(* PLC project BASIC, CODESYS CODESYS V3.5 SP16, author oscat *)
(* stored: creationDateTime 2020-05-24T16:39:18.0227817, version 3.31, modificationDateTime 2020-05-03T13:16:44.3823838, organization OSCAT *)
(* www.oscat.de *)

TYPE CALENDAR : STRUCT
  UTC : DT;  (* world time UTC *)
  YEAR : INT;  (* year of LDATE *)
  MONTH : INT;  (* month of LDATE *)
  DAY : INT;  (* day of LDATE *)
  WEEKDAY : INT;  (* weekday of LDATE *)
  OFFSET : INT;  (* Time Zone Offset for Local time in minutes *)
  DST_EN : BOOL;  (* daylight savings time enable *)
  DST_ON : BOOL;  (* true when daylight savings time os on *)
  NAME : STRING(5);  (* name of time zone *)
  LANGUAGE : INT;  (* location number pls see location setup *)
  LONGITUDE : REAL;  (* longitude of current location *)
  LATITUDE : REAL;  (* latitude of current location *)
  SUN_RISE : TOD;  (* sun_rise for current location *)
  SUN_SET : TOD;  (* sun_set for current location *)
  SUN_MIDDAY : TOD;  (* worldtime when sun stands at south position *)
  SUN_HEIGTH : REAL;  (* suns heigth at midday, south position *)
  SUN_HOR : REAL;  (* sun angle horizontal 0 = north in degrees *)
  SUN_VER : REAL;  (* sun angle vertical above horizon in degrees *)
  NIGHT : BOOL;  (* true between sun_set and sun_rise *)
  HOLIDAY : BOOL;  (* true when holiday *)
  HOLY_NAME : STRING(30);  (* name of holiday *)
  WORK_WEEK : INT;  (* current work week *)
END_STRUCT;
END_TYPE

TYPE COMPLEX : STRUCT
  re : REAL;
  im : REAL;
END_STRUCT;
END_TYPE

TYPE CONSTANTS_LANGUAGE : STRUCT
  DEFAULT : INT := 1;  (* 1=english, 2=german 3=french *)
  LMAX : INT := 3;
  WEEKDAYS : ARRAY[1..3, 1..7] OF STRING(10) := ['Monday', 'Tuesday', 'Wednesday', 'Thursday', 'Friday', 'Saturday', 'Sunday', 'Montag', 'Dienstag', 'Mittwoch', 'Donnerstag', 'Freitag', 'Samstag', 'Sonntag', 'Lundi', 'Mardi', 'Mercredi', 'Jeudi', 'Vendredi', 'Samedi', 'Dimanche'];
  WEEKDAYS2 : ARRAY[1..3, 1..7] OF STRING(2) := ['Mo', 'Tu', 'We', 'Th', 'Fr', 'Sa', 'Su', 'Mo', 'Di', 'Mi', 'Do', 'Fr', 'Sa', 'So', 'Lu', 'Ma', 'Me', 'Je', 'Ve', 'Sa', 'Di'];
  MONTHS : ARRAY[1..3, 1..12] OF STRING(10) := ['January', 'February', 'March', 'April', 'May', 'June', 'July', 'August', 'September', 'October', 'November', 'December', 'Januar', 'Februar', 'März', 'April', 'Mai', 'Juni', 'Juli', 'August', 'September', 'Oktober', 'November', 'Dezember', 'Janvier', 'Février', 'mars', 'Avril', 'Mai', 'Juin', 'Juillet', 'Août', 'Septembre', 'Octobre', 'Novembre', 'Decembre'];
  MONTHS3 : ARRAY[1..3, 1..12] OF STRING(3) := ['Jan', 'Feb', 'Mar', 'Apr', 'May', 'Jun', 'Jul', 'Aug', 'Sep', 'Oct', 'Nov', 'Dec', 'Jan', 'Feb', 'Mrz', 'Apr', 'Mai', 'Jun', 'Jul', 'Aug', 'Sep', 'Okt', 'Nov', 'Dez', 'Jan', 'Fev', 'Mar', 'Avr', 'Mai', 'Jun', 'Jul', 'Aou', 'Sep', 'Oct', 'Nov', 'Dec'];
  DIRS : ARRAY[1..3, 0..15] OF STRING(3) := ['N', 'NNE', 'NE', 'ENE', 'E', 'ESE', 'SE', 'SSE', 'S', 'SSW', 'SW', 'WSW', 'W', 'WNW', 'NW', 'NNW', 'N', 'NNO', 'NO', 'ONO', 'O', 'OSO', 'SO', 'SSO', 'S', 'SSW', 'SW', 'WSW', 'W', 'WNW', 'NW', 'NNW', 'N', 'NNO', 'NO', 'ONO', 'O', 'OSO', 'SO', 'SSO', 'S', 'SSW', 'SW', 'WSW', 'W', 'WNW', 'NW', 'NNW'];
END_STRUCT;
END_TYPE

TYPE CONSTANTS_LOCATION : STRUCT
  DEFAULT : INT := 1;  (* 1=germany, 2=austria 3=france 4=belgium-german 5= italien-Südtirol *)
  LMAX : INT := 5;
  LANGUAGE : ARRAY[1..5] OF INT := [2, 2, 3, 2, 2];  (* language spoken in the location *)
END_STRUCT;
END_TYPE

TYPE CONSTANTS_MATH : STRUCT
  PI : REAL := 3.1415926535897931;  (* Kreiszahl PI *)
  PI2 : REAL := 6.2831853071795862;  (* PI * 2 *)
  PI4 : REAL := 12.566370614359172;  (* PI * 4 *)
  PI05 : REAL := 1.5707963267949;  (* PI / 2 *)
  PI025 : REAL := 0.785398163397448;  (* PI / 4 *)
  PI_INV : REAL := 0.318309886183791;  (* 1 / PI *)
  E : REAL := 2.7182818284590451;  (* Eulersche Konstante e *)
  E_INV : REAL := 0.367879441171442;  (* 1 / e *)
  SQ2 : REAL := 1.4142135623731;  (* Wurzel von 2 *)
END_STRUCT;
END_TYPE

TYPE CONSTANTS_PHYS : STRUCT
  C : REAL := 299792458;  (* Lichtgeschwindigkeit in m/s *)
  E : REAL := 1.60217653E-19;  (* elementarladung in Colomb = A * s *)
  G : REAL := 9.80665;  (* Erdbeschleunigung in m / s² *)
  T0 : REAL := -273.15;  (* absoluter Nullpunkt in °C *)
  RU : REAL := 8.314472;  (* Universelle Gaskonstante in J / (mol · K) *)
  PN : REAL := 101325;  (* NormalDruck in Pa *)
END_STRUCT;
END_TYPE

TYPE CONSTANTS_SETUP : STRUCT
  EXTENDED_ASCII : BOOL := TRUE;  (* setup Parameters *)
  CHARNAMES : ARRAY[1..4] OF STRING(253) := [';"&quot;&&amp;<&lt;>&gt;&euro; &nbsp;¡&iexcl;¢&cent;£&pound;¤&curren;¥&yen;¦&brvbar;§&sect;¨&uml;©&copy;ª&ordf;«&laquo;¬&not;­&shy;®&reg;¯&macr;°&deg;±&plusmn;²&sup2;³&sup3;´&acute;µ&micro;¶&para;·&middot;¸&cedil;¹&sup1;º&ordm;»&raquo;¼&frac14;Û&Ucirc;', ';¾&frac34;¿&iquest;À&Agrave;Á&Aacute;Â&Acirc;Ã&Atilde;Ä&Auml;Å&Aring;Æ&AElig;Ç&Ccedil;È&Egrave;É&Eacute;Ê&Ecirc;Ë&Euml;Ì&Igrave;Í&Iacute;Î&Icirc;Ï&Iuml;Ð&ETH;Ñ&Ntilde;Ò&Ograve;Ó&Oacute;Ô&Ocirc;Õ&Otilde;Ö&Ouml;×&times;Ø&Oslash;Ù&Ugrave;Ú&Uacute;½&frac12;', ';Ü&Uuml;Ý&Yacute;Þ&THORN;ß&szlig;à&agrave;á&aacute;â&acirc;ã&atilde;ä&auml;å&aring;æ&aelig;ç&ccedil;è&egrave;é&eacute;ê&ecirc;ë&euml;ì&igrave;í&iacute;î&icirc;ï&iuml;ð&eth;ñ&ntilde;ò&ograve;ó&oacute;ô&ocirc;õ&otilde;ö&ouml;÷&divide;ø&oslash;ù&ugrave;', ';ú&uacute;û&ucirc;ü&uuml;ý&yacute;þ&thorn;ÿ&yuml;'];
  MTH_OFS : ARRAY[1..12] OF INT := [0, 31, 59, 90, 120, 151, 181, 212, 243, 273, 304, 334];
  DECADES : ARRAY[0..8] OF REAL := [1, 10, 100, 1000, 10000, 10000, 100000, 1000000, 10000000];
END_STRUCT;
END_TYPE

TYPE ESR_DATA : STRUCT
  TYP : BYTE;
  ADRESS : STRING(10);
  DS : DT;
  TS : TIME;
  DATA : ARRAY[0..7] OF BYTE;
END_STRUCT;
END_TYPE

TYPE FRACTION : STRUCT
  NUMERATOR : INT;
  DENOMINATOR : INT;
END_STRUCT;
END_TYPE

TYPE HOLIDAY_DATA : STRUCT
  NAME : STRING(30);
  DAY : SINT;
  MONTH : SINT;
  USE : SINT;
END_STRUCT;
END_TYPE

TYPE REAL2 : STRUCT
  R1 : REAL;  (* small value *)
  RX : REAL;  (* big value *)
END_STRUCT;
END_TYPE

TYPE SDT : STRUCT
  YEAR : INT;
  MONTH : INT;
  DAY : INT;
  WEEKDAY : INT;
  HOUR : INT;
  MINUTE : INT;
  SECOND : INT;
  MS : INT;
END_STRUCT;
END_TYPE

TYPE TIMER_EVENT : STRUCT
  TYP : BYTE;
  CHANNEL : BYTE;
  DAY : BYTE;
  START : TOD;
  DURATION : TIME;
  LAND : BYTE;
  LOR : BYTE;
  LAST : DT;
END_STRUCT;
END_TYPE

TYPE VECTOR_3 : STRUCT
  X : REAL;
  Y : REAL;
  Z : REAL;
END_STRUCT;
END_TYPE

VAR_GLOBAL CONSTANT  (* Constants *)
  STRING_LENGTH : INT := 250;
  LIST_LENGTH : INT := 250;
END_VAR

VAR_GLOBAL  (* Globale_Variablen *)
  MATH : CONSTANTS_MATH;
  PHYS : CONSTANTS_PHYS;
  LANGUAGE : CONSTANTS_LANGUAGE;
  SETUP : CONSTANTS_SETUP;
  LOCATION : CONSTANTS_LOCATION;
END_VAR


FUNCTION _BUFFER_CLEAR : BOOL
  VAR_INPUT
    PT : POINTER TO BYTE;
    SIZE : UINT;
  END_VAR
  VAR
    ptw : POINTER TO DWORD;
    temp : DWORD;
    end : DWORD;
    end32 : DWORD;
  END_VAR

            (* this routine uses 32 bit access to gain speed *)
(* first access bytes till pointer is aligned for 32 bit access *)
temp := pt;
end := temp + UINT_TO_DWORD(size);
end32 := end - 3;
WHILE (pt < end) AND ((temp AND 16#00000003) > 0) DO
	pt^ := 0;
	pt := pt + 1;
	temp := temp + 1;
END_WHILE;
(* pointer is aligned, now copy 32 bits at a time *)
ptw := pt;
WHILE ptw < end32 DO (* *)
	ptw^ := 0;
	ptw := ptw + 4;
END_WHILE;
(* copy the remaining bytes in byte mode *)
pt := ptw;
WHILE pt < end DO
	pt^ := 0;
	pt := pt + 1;
END_WHILE;

_BUFFER_CLEAR := TRUE;

(* revision History
hm 	5. mar. 2008	rev 1.0
	original version

hm	16. mar. 2008	rev 1.1
	added type conversion to avoid warnings under codesys 30
	chaged type of input size to uint
	deleted unused variable i

hm	31. oct. 2008	rev 1.2
	corrected an error while routine would write outside of arrays

*)
          
END_FUNCTION

FUNCTION _BUFFER_INIT : BOOL
  VAR_INPUT
    PT : POINTER TO BYTE;
    SIZE : UINT;
    INIT : BYTE;
  END_VAR
  VAR
    ptw : POINTER TO DWORD;
    temp : DWORD;
    end : DWORD;
    end32 : DWORD;
  END_VAR

            (* this routine uses 32 bit access to gain speed *)
(* first access bytes till pointer is aligned for 32 bit access *)
temp := pt;
end := temp + UINT_TO_DWORD(size);
end32 := end - 3;
WHILE (pt < end) AND ((temp AND 16#00000003) > 0) DO
	pt^ := init;
	pt := pt + 1;
	temp := temp + 1;
END_WHILE;
(* pointer is aligned, now copy 32 bits at a time *)
ptw := pt;
temp := SHL(BYTE_TO_DWORD(init),24) OR SHL(BYTE_TO_DWORD(init),16) OR SHL(BYTE_TO_DWORD(init),8) OR BYTE_TO_DWORD(init);
WHILE ptw < end32 DO
	ptw^ := temp;
	ptw := ptw + 4;
END_WHILE;
(* copy the remaining bytes in byte mode *)
pt := ptw;
WHILE pt < end DO
	pt^ := init;
	pt := pt + 1;
END_WHILE;

_BUFFER_INIT := TRUE;

(* revision History
hm 	5. mar. 2008	rev 1.0
	original version

hm	16. mar. 2008	rev 1.1
	added type conversion to avoid warnings under codesys 3.0
	chaged type of input size to uint.

hm	31. oct. 2008	rev 1.2
	corrected an error while routine would write outside of arrays

*)
          
END_FUNCTION

FUNCTION _BUFFER_INSERT : BOOL
  VAR_INPUT
    STR : STRING(STRING_LENGTH);
    POS : INT;
    PT : POINTER TO ARRAY[0..32767] OF BYTE;
    SIZE : UINT;
  END_VAR
  VAR
    end : INT;
    lx : INT;
    i : INT;
  END_VAR

            lx := LEN(str);
end := pos + lx;
(* first move the upper part of the buffer to make space for the string *)
FOR i := UINT_TO_INT(size) - 1 TO end BY -1 DO
	pt^[i] := pt^[i-lx];
END_FOR;
(* copy the string *)
_BUFFER_INSERT := _STRING_TO_BUFFER(str, pos, PT, size);


(* revision History
hm 	9. mar. 2008	rev 1.0
	original version

hm	16. mar. 2008	rev 1.1
	changed type of input size to uint

hm	13. may. 2008	rev 1.2
	changed type of pointer to array[1..32767]
	changed size of string to STRING_LENGTH

hm	23. mar. 2009	rev 1.3
	avoid writing to input pos

hm	12. nov. 2009	rev 1.4
	code optimized

*)
          
END_FUNCTION

FUNCTION _BUFFER_UPPERCASE : BOOL
  VAR_INPUT
    PT : POINTER TO ARRAY[0..32000] OF BYTE;
    SIZE : INT;
  END_VAR
  VAR
    pos : INT;
  END_VAR

            pos := 0;
WHILE pos < size DO
	PT^[pos] := TO_UPPER(pt^[pos]);
	pos := pos + 1;
END_WHILE;

_BUFFER_UPPERCASE := TRUE;

(* revision History
hm 	20. jan. 2011	rev 1.0
	original version

*)
          
END_FUNCTION

FUNCTION _STRING_TO_BUFFER : BOOL
  VAR_INPUT
    STR : STRING(STRING_LENGTH);
    POS : INT;
    PT : POINTER TO ARRAY[0..32767] OF BYTE;
    SIZE : UINT;
  END_VAR
  VAR
    ps : POINTER TO BYTE;
    i : INT;
    end : INT;
  END_VAR

            ps := ADR(str);
end := MIN(pos + LEN(str), UINT_TO_INT(size));
IF end > 0 THEN end := end -1; END_IF;
FOR i := pos TO end DO
	pt^[i] := ps^;
	ps := ps + 1;
END_FOR;

_STRING_TO_BUFFER := TRUE;

(* revision History

hm 	5. mar. 2008	rev 1.0
	original version

hm	16. mar. 2008	rev 1.1
	changed type of input size to uint

hm	13. may. 2008	rev 1.2
	changed type of pointer to array[1..32767]
	changed size of string to STRING_LENGTH

hm	12. nov. 2009	rev 1.3
	limit end to size - 1

*)
          
END_FUNCTION

FUNCTION BUFFER_COMP : INT
  VAR_INPUT
    PT1 : POINTER TO ARRAY[0..32767] OF BYTE;
    SIZE1 : INT;
    PT2 : POINTER TO ARRAY[0..32767] OF BYTE;
    SIZE2 : INT;
    START : INT;
  END_VAR
  VAR
    i : INT;
    j : INT;
    end : INT;
    firstbyte : BYTE;
  END_VAR

            (* search for first character match *)
IF size2 <= size1 THEN
	end := size1 - size2;
	firstbyte := PT2^[0];
	FOR i := START TO end DO
		IF PT1^[i] = firstbyte THEN
			(* first character matches, now compare rest of array *)
			j := 1;
			WHILE j < size2 DO
				IF pt2^[j] <> pt1^[j+i] THEN EXIT; END_IF;
				j := j + 1;
			END_WHILE;
			(* when J > size2 a match was found return the position i in buffer1 *)
			IF j = size2 THEN
				BUFFER_COMP := i;
				RETURN;
			END_IF;
		END_IF;
	END_FOR;
END_IF;
BUFFER_COMP := -1;


(*
hm 14. nov. 2008	rev 1.0
	original version

hm	12. nov. 2009	rev 1.1
	performance increase

*)
          
END_FUNCTION

FUNCTION BUFFER_SEARCH : INT
  VAR_INPUT
    PT : POINTER TO ARRAY[0..32767] OF BYTE;
    SIZE : INT;
    STR : STRING(STRING_LENGTH);
    POS : INT;
    IGN : BOOL;
  END_VAR
  VAR
    ps : POINTER TO ARRAY[0..STRING_LENGTH] OF BYTE;
    chx : BYTE;
    i : INT;
    end : INT;
    k : INT;
    lx : INT;
  END_VAR

            ps := ADR(STR);
lx := LEN(STR);
end := MIN(SIZE - lx, SIZE - 1);
lx := lx - 1;
FOR i := pos TO end DO
	FOR k := 0 TO lx DO
		IF IGN THEN chx := TO_UPPER(pt^[i+k]); ELSE chx := pt^[i+k]; END_IF;
		IF ps^[k] <> chx THEN EXIT; END_IF;
	END_FOR;
	IF k > lx THEN
		BUFFER_SEARCH := i;
		RETURN;
	END_IF;
END_FOR;
BUFFER_SEARCH := -1;


(* revision History

hm 5. mar. 2008	rev 1.0
	original version

hm	16. mar. 2008	rev 1.1
	chaged type of input size to uint

hm	13. may. 2008	rev 1.2
	changed type of pointer to array[1..32767]
	changed size of string to STRING_LENGTH

hm	12. nov. 2009	rev 1.3
	limit end to array size

hm	25. jan. 2011	rev 1.4
	ign = True will now ignore case
	return -1 if nothing found
*)
          
END_FUNCTION

FUNCTION BUFFER_TO_STRING : STRING(STRING_LENGTH)
  VAR_INPUT
    PT : POINTER TO ARRAY[0..32767] OF BYTE;
    SIZE : UINT;
    START : UINT;
    STOP : UINT;
  END_VAR
  VAR
    ps : POINTER TO BYTE;
    i : UINT;
    stp : UINT;
    sta : UINT;
  END_VAR

            ps := ADR(BUFFER_TO_STRING);
IF size = 0 THEN RETURN; END_IF;
sta := MIN(start, size -1);
stp := MIN(stop, size -1);

(* check for maximum string_length *)
IF UINT_TO_INT(stp - sta + 1) >= STRING_LENGTH THEN
	stp := sta + INT_TO_UINT(STRING_LENGTH) - 1;
END_IF;

FOR i := sta TO stp DO
	ps^ := pt^[i];
	ps := ps + 1;
END_FOR;

(* terminate the string *)

ps^ := 0;



(* revision History
hm 	5. mar. 2008	rev 1.0
	original version

hm	16. mar. 2008	rev 1.1
	changed type of input size to uint

hm	13. may. 2008	rev 1.2
	changed type of pointer to array[0..32767]
	changed size of string to STRING_LENGTH

hm	12. jun. 2008	rev 1.3
	check for pointer overrun
	change input start and stop to uint
	added type conversions to avoid warnings under codesys 3.0

hm	23. mar. 2009	rev 1.4
	avoid writing to input stop

hm	12. nov. 2009 rev 1.5
	limit start and stop to size -1

*)
          
END_FUNCTION

FUNCTION_BLOCK DRIVER_1
  VAR_INPUT
    {attribute 'input_constant'}
    Toggle_Mode : BOOL;
    {attribute 'input_constant'}
    Timeout : TIME;
    SET : BOOL;
    IN : BOOL;
    RST : BOOL;
  END_VAR
  VAR_OUTPUT
    Q : BOOL;
  END_VAR
  VAR
    off : TON;
    edge : BOOL;
  END_VAR

            IF off.Q THEN Q := FALSE; END_IF;
IF rst THEN
	Q := FALSE;
ELSIF set THEN
	Q := TRUE;
ELSIF IN AND NOT edge THEN
	IF toggle_mode THEN q := NOT Q; ELSE q := TRUE; END_IF;
END_IF;
edge := in;
IF timeout > t#0s THEN off(in := Q, PT := Timeout); END_IF;


(* revision history
hm	2. jan 2008		rev 1.0
	original version

*)
          
END_FUNCTION_BLOCK

FUNCTION_BLOCK DRIVER_4
  VAR_INPUT
    {attribute 'input_constant'}
    Toggle_Mode : BOOL;
    {attribute 'input_constant'}
    Timeout : TIME;
    SET : BOOL;
    IN0 : BOOL;
    IN1 : BOOL;
    IN2 : BOOL;
    IN3 : BOOL;
    RST : BOOL;
  END_VAR
  VAR_OUTPUT
    Q0 : BOOL;
    Q1 : BOOL;
    Q2 : BOOL;
    Q3 : BOOL;
  END_VAR
  VAR
    d0 : DRIVER_1;
    d1 : DRIVER_1;
    d2 : DRIVER_1;
    d3 : DRIVER_1;
  END_VAR

            D0(Set:=set, in:=in0, rst:=rst, toggle_mode:=toggle_mode, timeout:=timeout);
D1(Set:=set, in:=in1, rst:=rst, toggle_mode:=toggle_mode, timeout:=timeout);
D2(Set:=set, in:=in2, rst:=rst, toggle_mode:=toggle_mode, timeout:=timeout);
D3(Set:=set, in:=in3, rst:=rst, toggle_mode:=toggle_mode, timeout:=timeout);
Q0 := D0.Q;
Q1 := D1.Q;
Q2 := D2.Q;
Q3 := D3.Q;


(* revision history
hm	2. jan 2008		rev 1.0
	original version

*)
          
END_FUNCTION_BLOCK

FUNCTION_BLOCK DRIVER_4C
  VAR_INPUT
    IN : BOOL;
    RST : BOOL;
    {attribute 'input_constant'}
    Timeout : TIME;
    {attribute 'input_constant'}
    SX : ARRAY[1..7] OF BYTE := [1, 3, 7, 15];
  END_VAR
  VAR_OUTPUT
    SN : INT;
    Q0 : BOOL;
    Q1 : BOOL;
    Q2 : BOOL;
    Q3 : BOOL;
  END_VAR
  VAR
    off : TON;
    edge : BOOL;
  END_VAR

            IF RST OR off.Q THEN
	SN := 0;
ELSIF IN AND NOT edge THEN
	SN := SN + 1;
	IF SN > 7 OR SX[SN] = 0 THEN SN := 0; END_IF;
END_IF;
edge := in;
IF SN > 0 THEN
	Q0 := SX[SN].0;
	Q1 := SX[SN].1;
	Q2 := SX[SN].2;
	Q3 := SX[SN].3;
ELSE
	Q0 := FALSE;
	Q1 := FALSE;
	Q2 := FALSE;
	Q3 := FALSE;
END_IF;

(* maximaum timeout *)
IF timeout > t#0s THEN off(in := SN > 0, PT := Timeout); END_IF;


(* revision history
hm	23. mar. 2009	rev 1.0
	original version

*)
          
END_FUNCTION_BLOCK

FUNCTION_BLOCK FLOW_CONTROL
  VAR_INPUT
    IN : BOOL;
    REQ : BOOL;
    ENQ : BOOL;
    RST : BOOL;
    {attribute 'input_constant'}
    T_AUTO : TIME := TIME#60m0s0ms;
    {attribute 'input_constant'}
    T_DELAY : TIME := TIME#1380m0s0ms;
  END_VAR
  VAR_OUTPUT
    Q : BOOL;
    STATUS : BYTE;
  END_VAR
  VAR
    timer : TP_1D;
  END_VAR

            STATUS := 100;
IF RST THEN
	Q := FALSE;
	timer(rst := TRUE);
	timer.RST := FALSE;
	STATUS := 103;
ELSIF ENQ THEN
	IF IN THEN
		status := 101;
	END_IF;
	IF REQ THEN
		(* timer will generate a timed pulse after TP goes high *)
		timer.PT1 := T_AUTO;
		timer.PTD := T_DELAY;
		timer.IN := TRUE;
		STATUS := 102;
	END_IF;
END_IF;


(* set output and run timer *)
timer();
timer.IN := FALSE;
Q := (IN AND ENQ) OR timer.Q;



(* revision history
hm 	28. jun. 2008 	rev 1.0
	original version

*)
          
END_FUNCTION_BLOCK

FUNCTION_BLOCK FT_Profile
  VAR_INPUT
    K : REAL := 1;
    O : REAL;
    M : REAL := 1;
    E : BOOL;
    {attribute 'input_constant'}
    value_0 : REAL;
    {attribute 'input_constant'}
    time_1 : TIME;
    {attribute 'input_constant'}
    value_1 : REAL;
    {attribute 'input_constant'}
    time_2 : TIME;
    {attribute 'input_constant'}
    value_2 : REAL;
    {attribute 'input_constant'}
    time_3 : TIME;
    {attribute 'input_constant'}
    value_3 : REAL;
    {attribute 'input_constant'}
    time_10 : TIME;
    {attribute 'input_constant'}
    value_10 : REAL;
    {attribute 'input_constant'}
    time_11 : TIME;
    {attribute 'input_constant'}
    value_11 : REAL;
    {attribute 'input_constant'}
    time_12 : TIME;
    {attribute 'input_constant'}
    value_12 : REAL;
    {attribute 'input_constant'}
    time_13 : TIME;
    {attribute 'input_constant'}
    value_13 : REAL;
  END_VAR
  VAR_OUTPUT
    Y : REAL;
    RUN : BOOL;
    ET : TIME;
  END_VAR
  VAR
    tx : TIME;
    edge : BOOL;
    state : BYTE;
    ta : TIME;
    tb : TIME;
    t0 : TIME;
    temp : REAL;
    va : REAL;
    vb : REAL;
  END_VAR

            (* read system time *)
tx := DWORD_TO_TIME(T_PLC_MS());

(* determine start condition *)
IF E AND NOT edge THEN
	RUN := TRUE;
	ET := t#0s;
	t0 := tx;
	ta := tx;
	tb := multime(time_1, M);
	va := value_0;
	vb := value_1;
	temp := value_0;
	state := 1;
END_IF;
edge := E;

(* generate startup profile *)
IF run THEN
	CASE state OF
		1:	IF tx - ta >= tb THEN
				ta := ta + tb;
				tb := multime(time_2 - time_1, M);
				va := value_1;
				vb := value_2;
				temp := value_1;
				state := 2;
			ELSE
				temp := ((vb - va) * TIME_TO_REAL(tx - ta) / TIME_TO_REAL(tb) + va);
			END_IF;
		2:	IF tx - ta >= tb THEN
				ta := ta + tb;
				tb := multime(time_3 - time_2, M);
				va := value_2;
				vb := value_3;
				temp := value_2;
				state := 3;
			ELSE
				temp := ((vb - va) * TIME_TO_REAL(tx - ta) / TIME_TO_REAL(tb) + va);
			END_IF;
		3:	IF tx - ta >= tb THEN
				ta := ta + tb;
				tb := multime(time_10 - time_3, M);
				va := value_3;
				vb := value_10;
				temp := value_3;
				state := 4;
			ELSE
				temp := ((vb - va) * TIME_TO_REAL(tx - ta) / TIME_TO_REAL(tb) + va);
			END_IF;
		4 :	IF tx - ta >= tb THEN
				ta := ta + tb;
				tb := multime(time_11 - time_10, M);
				va := value_10;
				vb := value_11;
				temp := value_10;
				IF E THEN state := 5; ELSE state := 6; END_IF;
			ELSE
				temp := ((vb - va) * TIME_TO_REAL(tx - ta) / TIME_TO_REAL(tb) + va);
			END_IF;
		5:	(* extend the signal while E is true *)
			IF E THEN
				ta := tx;
			ELSE
				state := 6;
			END_IF;
		6:	IF tx - ta >= tb THEN
				ta := ta + tb;
				tb := multime(time_12 - time_11, M);
				va := value_11;
				vb := value_12;
				temp := value_11;
				state := 7;
			ELSE
				temp := ((vb - va) * TIME_TO_REAL(tx - ta) / TIME_TO_REAL(tb) + va);
			END_IF;
		7:	IF tx - ta >= tb THEN
				ta := ta + tb;
				tb := multime(time_13 - time_12, M);
				va := value_12;
				vb := value_13;
				temp := value_12;
				state := 8;
			ELSE
				temp := ((vb - va) * TIME_TO_REAL(tx - ta) / TIME_TO_REAL(tb) + va);
			END_IF;
		8:	IF tx - ta >= tb THEN
				temp := value_13;
				run := FALSE;
			ELSE
				temp := ((vb - va) * TIME_TO_REAL(tx - ta) / TIME_TO_REAL(tb) + va);
			END_IF;
	END_CASE;
	Y := temp * K + O;
	ET := tx - t0;
END_IF;

(* revision history
hm	27 feb 2007		rev 1.0
	original version

hm	15. sep2007		rev 1.1
	replaced Time() with T_PLC_MS for compatibility and performance reasons

*)
          
END_FUNCTION_BLOCK

FUNCTION_BLOCK INC_DEC
  VAR_INPUT
    CHa : BOOL;
    CHb : BOOL;
    RST : BOOL;
  END_VAR
  VAR_OUTPUT
    dir : BOOL;
    cnt : INT;
  END_VAR
  VAR
    edgea : BOOL;
    clk : BOOL;
    clka : BOOL;
    clkb : BOOL;
    edgeb : BOOL;
    axb : BOOL;
  END_VAR

            axb := cha XOR chb;

(* create pulses for channel a *)
clka := cha XOR edgea;
edgea := cha;

clkb := chb XOR edgeb;
edgeb := chb;

(* create pulses for both channels *)
clk := clka OR clkb;

(* set the direction output *)
IF axb AND clka THEN dir := TRUE; END_IF;
IF axb AND clkb THEN dir := FALSE; END_IF;

(* increment or decrement the counter *)
IF clk AND dir THEN cnt := cnt + 1; END_IF;
IF clk AND NOT dir THEN cnt := cnt -1; END_IF;

(* reset the counter if rst active *)
IF rst THEN cnt := 0; END_IF;

          
END_FUNCTION_BLOCK

FUNCTION_BLOCK INTERLOCK
  VAR_INPUT
    I1 : BOOL;
    I2 : BOOL;
    TL : TIME;
  END_VAR
  VAR_OUTPUT
    Q1 : BOOL;
    Q2 : BOOL;
  END_VAR
  VAR
    T1 : TOF;
    T2 : TOF;
  END_VAR

            (* the input signal have a run delay to lockout the other input *)
T1(IN := I1, PT := TL);
T2(IN := I2, PT := TL);

Q1 := I1 AND NOT t2.Q;
Q2 := I2 AND NOT t1.Q;


(* revision history

hm	28 sep 2007		rev 1.0
	original version

*)
          
END_FUNCTION_BLOCK

FUNCTION_BLOCK INTERLOCK_4
  VAR_INPUT
    I0 : BOOL;
    I1 : BOOL;
    I2 : BOOL;
    I3 : BOOL;
    E : BOOL;
    MODE : INT;
  END_VAR
  VAR_OUTPUT
    OUT : BYTE;
    TP : BOOL;
  END_VAR
  VAR
    in : BYTE;
    last : BYTE;
    old : BYTE;
    lmode : INT;
  END_VAR

            (* check if enable is active *)
IF E THEN
(* reset all vars when there is a mode change on thy fly *)
	IF mode <> lmode THEN
		out := 0;
		last := 0;
		old := 0;
		lmode := mode;
	END_IF;
	(* load inputs into in *)
	in.0 := I0;
	in.1 := I1;
	in.2 := I2;
	in.3 := I3;
	(* only execute when there is any change *)
	IF in <> last THEN
		(* only execute when inputs have chages state *)
		CASE mode OF
			0:	(* output directly display inputs as bits in byte out *)
				out := in;

			1:	(* the input with the highest number will be acepted *)
				IF in.3 THEN out := 8;
				ELSIF in.2 THEN out := 4;
				ELSIF in.1 THEN out := 2;
				ELSE out := in;
				END_IF;

			2:	(* input last pressed will be displayed only *)
				last := ((in XOR last) AND in);
				IF last.3 THEN out := 8;
				ELSIF last.2 THEN out := 4;
				ELSIF last.1 THEN out := 2;
				ELSE out := last;
				END_IF;

			3:	(* any input active will disable all other inputs *)
				IF (out AND in) = 0 THEN
					IF in.3 THEN out := 8;
					ELSIF in.2 THEN out := 4;
					ELSIF in.1 THEN out := 2;
					ELSE out := in;
					END_IF;
				END_IF;

		END_CASE;
		last := in;
	END_IF;
	tp := out <> old;
	old := out;
ELSE
	out := 0;
	last := 0;
	old := 0;
	lmode := 0;
	tp := FALSE;
END_IF;


(* revision history
hm	24. oct 2008	rev 1.0
	original version

hm	14. mar. 2009	rev 1.1
	replaced double assignments

*)
          
END_FUNCTION_BLOCK

FUNCTION MANUAL : BOOL
  VAR_INPUT
    IN : BOOL;
    ON : BOOL;
    OFF : BOOL;
  END_VAR

            MANUAL := NOT OFF AND (IN OR ON);



(* revision history
hm	21. nov 2008	rev 1.0
	original version


*)
          
END_FUNCTION

FUNCTION_BLOCK MANUAL_1
  VAR_INPUT
    IN : BOOL;
    MAN : BOOL;
    M_I : BOOL;
    SET : BOOL;
    RST : BOOL;
  END_VAR
  VAR_OUTPUT
    Q : BOOL;
    STATUS : BYTE;
  END_VAR
  VAR
    S_edge : BOOL;
    r_edge : BOOL;
    edge : BOOL;
  END_VAR

            IF NOT man THEN
	Q := IN;
	STATUS := 100;
	edge := FALSE;
ELSIF NOT s_edge AND set THEN
	Q := TRUE;
	edge := TRUE;
	status := 101;
ELSIF NOT r_edge AND rst THEN
	Q := FALSE;
	edge := TRUE;
	status := 102;
ELSIF NOT edge THEN
	Q := M_I;
	status := 103;
END_IF;

(* remember levels of manual signals *)
s_edge := SET;
r_edge := RST;



(* revision history
hm	17. jun 2008	rev 1.0
	original version

hm	17. oct 2008	rev 1.1
	deleted unnecessary variable m_edge

hm	14. mar. 2009	rev 1.2
	replaced double assignments

*)
          
END_FUNCTION_BLOCK

FUNCTION_BLOCK MANUAL_2
  VAR_INPUT
    IN : BOOL;
    ENA : BOOL;
    ON : BOOL;
    OFF : BOOL;
    MAN : BOOL;
  END_VAR
  VAR_OUTPUT
    Q : BOOL;
    STATUS : BYTE;
  END_VAR

            IF ena THEN
	IF NOT ON AND NOT OFF THEN
		Q := IN;
		STATUS := 100;
	ELSIF on AND NOT off THEN
		Q := TRUE;
		STATUS := 101;
	ELSIF NOT on AND off THEN
		q := FALSE;
		STATUS := 102;
	ELSE
		Q := MAN;
		STATUS := 103;
	END_IF;
ELSE
	Q := FALSE;
	STATUS := 104;
END_IF;



(* revision history
hm	22. sep. 2008		rev 1.0
	original version

*)
          
END_FUNCTION_BLOCK

FUNCTION_BLOCK MANUAL_4
  VAR_INPUT
    I0 : BOOL;
    I1 : BOOL;
    I2 : BOOL;
    I3 : BOOL;
    MAN : BOOL;
    STP : BOOL;
    M0 : BOOL;
    M1 : BOOL;
    M2 : BOOL;
    M3 : BOOL;
  END_VAR
  VAR_OUTPUT
    Q0 : BOOL;
    Q1 : BOOL;
    Q2 : BOOL;
    Q3 : BOOL;
    STATUS : BYTE;
  END_VAR
  VAR
    edge : BOOL;
    pos : INT;
    tog : BOOL;
  END_VAR

            IF man THEN
	IF NOT TOG THEN
		Q0 := M0;
		Q1 := M1;
		Q2 := M2;
		Q3 := M3;
		STATUS := 101;
	END_IF;
	IF STP AND NOT edge THEN
		tog := TRUE;
		CASE pos OF
			0:	Q0 := TRUE;
				Q1 := FALSE;
				Q2 := FALSE;
				Q3 := FALSE;
				STATUS := 110;
			1:	Q0 := FALSE;
				Q1 := TRUE;
				Q2 := FALSE;
				Q3 := FALSE;
				STATUS := 111;
			2:	Q0 := FALSE;
				Q1 := FALSE;
				Q2 := TRUE;
				Q3 := FALSE;
				STATUS := 112;
			3:	Q0 := FALSE;
				Q1 := FALSE;
				Q2 := FALSE;
				Q3 := TRUE;
				STATUS := 113;
		END_CASE;
		pos := INC(pos,1,3);
	END_IF;
ELSE
	Q0 := I0;
	Q1 := I1;
	Q2 := I2;
	Q3 := I3;
	STATUS := 100;
	tog := FALSE;
	pos := 0;
END_IF;

(* remember status of stp *)
edge := STP;



(* revision history
hm	17. jun 2008		rev 1.0
	original version

*)
          
END_FUNCTION_BLOCK

FUNCTION_BLOCK PARSET
  VAR_INPUT
    A0 : BOOL;
    A1 : BOOL;
    {attribute 'input_constant'}
    X01 : REAL;
    {attribute 'input_constant'}
    X02 : REAL;
    {attribute 'input_constant'}
    X03 : REAL;
    {attribute 'input_constant'}
    X04 : REAL;
    {attribute 'input_constant'}
    X11 : REAL;
    {attribute 'input_constant'}
    X12 : REAL;
    {attribute 'input_constant'}
    X13 : REAL;
    {attribute 'input_constant'}
    X14 : REAL;
    {attribute 'input_constant'}
    X21 : REAL;
    {attribute 'input_constant'}
    X22 : REAL;
    {attribute 'input_constant'}
    X23 : REAL;
    {attribute 'input_constant'}
    X24 : REAL;
    {attribute 'input_constant'}
    X31 : REAL;
    {attribute 'input_constant'}
    X32 : REAL;
    {attribute 'input_constant'}
    X33 : REAL;
    {attribute 'input_constant'}
    X34 : REAL;
    {attribute 'input_constant'}
    TC : TIME;
  END_VAR
  VAR_OUTPUT
    P1 : REAL;
    P2 : REAL;
    P3 : REAL;
    P4 : REAL;
  END_VAR
  VAR
    X : ARRAY[0..3, 1..4] OF REAL;
    S1 : REAL;
    S2 : REAL;
    S3 : REAL;
    S4 : REAL;
    tx : DWORD;
    last : DWORD;
    start : BOOL;
    set : BYTE;
    init : BOOL;
  END_VAR

            (* read system_time *)
tx := T_PLC_MS();

(* init sequence *)
IF NOT init THEN
	set.0 := NOT A0;
	init := TRUE;
	X[0,1] := X01;
	X[0,2] := X02;
	X[0,3] := X03;
	X[0,4] := X04;
	X[1,1] := X11;
	X[1,2] := X12;
	X[1,3] := X13;
	X[1,4] := X14;
	X[2,1] := X21;
	X[2,2] := X22;
	X[2,3] := X23;
	X[2,4] := X24;
	X[3,1] := X31;
	X[3,2] := X32;
	X[3,3] := X33;
	X[3,4] := X34;
	P1 := X01;
	P2 := X02;
	P3 := X03;
	P4 := X04;
END_IF;

(* check for input change *)
IF (A0 XOR set.0) OR (A1 XOR set.1) THEN
	(* a new set is selected *)
	set.0 := A0;
	set.1 := A1;
	IF tc > t#0s THEN
		start := TRUE;
		last := tx;
		(* save the step speed for the output changes in S *)
		S1 := (X[set,1] - P1)/DWORD_TO_REAL(TIME_TO_DWORD(tc));
		S2 := (X[set,2] - P2)/DWORD_TO_REAL(TIME_TO_DWORD(tc));
		S3 := (X[set,3] - P3)/DWORD_TO_REAL(TIME_TO_DWORD(tc));
		S4 := (X[set,4] - P4)/DWORD_TO_REAL(TIME_TO_DWORD(tc));
	END_IF;
ELSIF start AND tx - last < TIME_TO_DWORD(tc) THEN
	(* ramp the outputs to the new value *)
	P1 := X[set,1] - S1 * DWORD_TO_REAL(TIME_TO_DWORD(Tc) - tx + last);
	P2 := X[set,2] - S2 * DWORD_TO_REAL(TIME_TO_DWORD(Tc) - tx + last);
	P3 := X[set,3] - S3 * DWORD_TO_REAL(TIME_TO_DWORD(Tc) - tx + last);
	P4 := X[set,4] - S4 * DWORD_TO_REAL(TIME_TO_DWORD(Tc) - tx + last);
ELSE
	(* make sure outputs match the correct set values *)
	start := FALSE;
	P1 := X[set,1];
	P2 := X[set,2];
	P3 := X[set,3];
	P4 := X[set,4];
END_IF;

(* revision history
hm	2.11.2007		rev 1.0
	original version

hm	16. mar. 2008	rev 1.1
	added type conversions to avoid warnings under codesys 3.0

*)

          
END_FUNCTION_BLOCK

FUNCTION_BLOCK PARSET2
  VAR_INPUT
    X : REAL;
    {attribute 'input_constant'}
    X01 : REAL;
    {attribute 'input_constant'}
    X02 : REAL;
    {attribute 'input_constant'}
    X03 : REAL;
    {attribute 'input_constant'}
    X04 : REAL;
    {attribute 'input_constant'}
    X11 : REAL;
    {attribute 'input_constant'}
    X12 : REAL;
    {attribute 'input_constant'}
    X13 : REAL;
    {attribute 'input_constant'}
    X14 : REAL;
    {attribute 'input_constant'}
    X21 : REAL;
    {attribute 'input_constant'}
    X22 : REAL;
    {attribute 'input_constant'}
    X23 : REAL;
    {attribute 'input_constant'}
    X24 : REAL;
    {attribute 'input_constant'}
    X31 : REAL;
    {attribute 'input_constant'}
    X32 : REAL;
    {attribute 'input_constant'}
    X33 : REAL;
    {attribute 'input_constant'}
    X34 : REAL;
    {attribute 'input_constant'}
    L1 : REAL;
    {attribute 'input_constant'}
    L2 : REAL;
    {attribute 'input_constant'}
    L3 : REAL;
    {attribute 'input_constant'}
    TC : TIME;
  END_VAR
  VAR_OUTPUT
    P1 : REAL;
    P2 : REAL;
    P3 : REAL;
    P4 : REAL;
  END_VAR
  VAR
    Pset : parset;
    init : BOOL;
  END_VAR

            (* init sequence *)
IF NOT init THEN
	init := TRUE;
	pset(TC:=TC, X01:=X01, X02:=X02, X03:=X03, X04:=X04, X11:=X11, X12:=X12, X13:=X13, X14:=X14, X21:=X21, X22:=X22, X23:=X23, X24:=X24, X31:=X31, X32:=X32, X33:=X33, X34:=X34);
END_IF;
IF ABS(X) < L1 THEN
	pset(A0 := FALSE, A1 := FALSE);
ELSIF ABS(X) < L2 THEN
	pset(A0 := TRUE, A1 := FALSE);
ELSIF ABS(x) < L3 THEN
	pset(A0 := FALSE, A1 := TRUE);
ELSE
	pset(A0 := TRUE, A1 := TRUE);
END_IF;
P1 := pset.P1;
P2 := pset.P2;
P3 := pset.P3;
P4 := pset.P4;

(* revision history
hm		3.11.2007		rev 1.0
	original version

*)

          
END_FUNCTION_BLOCK

FUNCTION_BLOCK SIGNAL
  VAR_INPUT
    IN : BOOL;
    SIG : BYTE;
    TS : TIME;
  END_VAR
  VAR_OUTPUT
    Q : BOOL;
  END_VAR
  VAR
    tx : DWORD;
    step : BYTE;
  END_VAR
  VAR CONSTANT
    one : BYTE := 1;
  END_VAR

            IF in THEN
	(* an alarm is present read system time first *)
	tx := T_PLC_MS();
	(* calculate the step counter which is the lowest 3 bits of (time / ts) *)
	IF ts > t#0s THEN
		step := DWORD_TO_BYTE(tx / TIME_TO_DWORD(ts) AND 16#0000_0007);
	ELSE
		step := DWORD_TO_BYTE(SHR(tx,7) AND 16#0000_0007);
	END_IF;
	(* convert the value 0-7 in step into one bit only (bit 0-7) *)
	step := SHL(one,step);
	(* generate the output signal *)
	Q := (step AND sig) > 0;
ELSE
	Q := FALSE;
END_IF;

(* revision history
hm	13.12.2007		rev 1.0
	original version

*)
          
END_FUNCTION_BLOCK

FUNCTION_BLOCK SIGNAL_4
  VAR_INPUT
    IN1 : BOOL;
    IN2 : BOOL;
    IN3 : BOOL;
    IN4 : BOOL;
    TS : TIME;
    {attribute 'input_constant'}
    S1 : BYTE := 2#11111111;
    {attribute 'input_constant'}
    S2 : BYTE := 2#11110000;
    {attribute 'input_constant'}
    S3 : BYTE := 2#10101010;
    {attribute 'input_constant'}
    S4 : BYTE := 2#10100000;
  END_VAR
  VAR_OUTPUT
    Q : BOOL;
  END_VAR
  VAR
    sig : SIGNAL;
  END_VAR

            (* an alarm is present read system time first *)
(* check if an alarm is present if yes set sig to the alarm pattern otherwise exit the routine *)
IF in1 THEN
	sig(in := TRUE, sig := s1, TS := TS);
ELSIF in2 THEN
	sig(in := TRUE, sig := s2, TS := TS);
ELSIF in3 THEN
	sig(in := TRUE, sig := s3, TS := TS);
ELSIF in4 THEN
	sig(in := TRUE, sig := s4, TS := TS);
ELSE
	sig(in := FALSE);
END_IF;

(* set the output *)
Q := sig.Q;


(* revision history
hm	13.12.2007		rev 1.0
	original version

*)

          
END_FUNCTION_BLOCK

FUNCTION_BLOCK SRAMP
  VAR_INPUT
    X : REAL;
    A_UP : REAL;
    A_DN : REAL;
    VU_MAX : REAL;
    VD_MAX : REAL;
    LIMIT_HIGH : REAL;
    LIMIT_LOW : REAL;
    RST : BOOL;
  END_VAR
  VAR_OUTPUT
    Y : REAL;
    V : REAL;
  END_VAR
  VAR
    cycle_time : TC_S;
    init : BOOL;
  END_VAR

            (* read the system_time in microseconds *)
cycle_time();

(* assure range of inputs *)
A_up := MAX(0.0, A_UP);
A_dn := MIN(0.0, A_dn);
VU_max := MAX(0.0, VU_max);
VD_max := MIN(0.0, VD_MAX);

(* calculate the output offset *)
IF rst OR NOT init THEN
	init := TRUE;
	Y := 0.0;
	V := 0.0;
ELSIF X = Y THEN
	v := 0.0;
ELSIF X > Y THEN
	(* output is too low >> ramp up and brake at the end *)
	(* accelerate the speed and limit to vu_max *)
	v := MIN(v + A_UP * cycle_time.TC, vu_max);
	(* calculate the max speed to be able to brake and select the lowest *)
	v := MIN(SQRT((Y-X) * 2.0 * A_DN), v);
	(* calculate the output and obey limits *)
	y := LIMIT(limit_low, y + MIN(v * cycle_time.TC, X-Y), limit_high);
ELSIF X < Y THEN
	(* output is too high >> ramp dn and brake at the end *)
	(* accelerate the speed and limit to vd_max *)
	v := MAX(v + A_DN * cycle_time.TC, vd_max);
	(* calculate the max speed to be able to brake and select the lowest *)
	v := MAX(-SQRT((Y-X) * 2.0 * A_UP), v);
	(* calculate the output and obey limits *)
	y := LIMIT(limit_low, y + MAX(v * cycle_time.TC, X-Y), limit_high);
END_IF;


(* revision history
hm	13. mar. 2008	rev 1.0
	original version

hm	11. mar. 2009	rev 1.1
	real constants updated to new systax using dot																																																																																																																																																																																																																																																																																																																																																																																																																																																																																																																																																																																																																																																																																																																																																																																																																																																																																																																																																																																																																																																											

*)



          
END_FUNCTION_BLOCK

FUNCTION_BLOCK TUNE
  VAR_INPUT
    SET : BOOL;
    SU : BOOL;
    SD : BOOL;
    RST : BOOL;
    {attribute 'input_constant'}
    SS : REAL := 0.1;
    {attribute 'input_constant'}
    Limit_L : REAL;
    {attribute 'input_constant'}
    LIMIT_H : REAL := 100;
    {attribute 'input_constant'}
    RST_val : REAL;
    {attribute 'input_constant'}
    SET_val : REAL := 100;
    {attribute 'input_constant'}
    T1 : TIME := TIME#500ms;
    {attribute 'input_constant'}
    T2 : TIME := TIME#2s0ms;
    {attribute 'input_constant'}
    S1 : REAL := 2;
    {attribute 'input_constant'}
    S2 : REAL := 10;
  END_VAR
  VAR_OUTPUT
    Y : REAL;
  END_VAR
  VAR
    tx : DWORD;
    start : DWORD;
    start2 : DWORD;
    state : INT;
    in : BOOL;
    step : REAL;
    SPEED : REAL;
    Y_start : REAL;
    Y_start2 : REAL;
  END_VAR

            (* read system time *)
tx := T_PLC_MS();

IF rst THEN
	Y := RST_val;
	state := 0;
ELSIF set THEN
	Y := SET_val;
	state := 0;
ELSIF state > 0 THEN
	(* key has been pushed state machine operating *)
	(* first read the correct input *)
	IF state = 1 THEN
		(* step up *)
		in := su;
	ELSE
		(* step down *)
		in := sd;
	END_IF;
	(* check for single step operation *)
	IF NOT in AND tx - start <= TIME_TO_DWORD(T1) THEN
		Y := Y_start + step;
		state := 0;
	(* check if fast ramp needs to be generated *)
	ELSIF in AND tx - start >= TIME_TO_DWORD(T2) THEN
		Y := Y_start2 + DWORD_TO_REAL(tx - start2) * s2 / speed;
	(* check if slow ramp needs to be generated *)
	ELSIF in AND tx - start >= TIME_TO_DWORD(T1) THEN
		Y := Y_start + DWORD_TO_REAL(tx - start - TIME_TO_DWORD(T1)) * S1 / speed;
		start2 := tx;
		Y_start2 := Y;
	ELSIF NOT in THEN
		state := 0;
	END_IF;
ELSIF su THEN
	(* slow step up *)
	state := 1;
	start := tx;
	step := ss;
	speed := 1000.0;
	Y_start := Y;
ELSIF sd THEN
	(* slow step down *)
	state := 2;
	start := tx;
	step := -ss;
	speed := -1000.0;
	Y_start := Y;
END_IF;

(* make sure output does not exceed limits *)
Y := LIMIT(LIMIT_L, Y, LIMIT_H);

(* revision history
hm	3.11.2007		rev 1.0
	original version

hm	16. mar. 2008	rev 1.1
	added type conversions to avoid warnings under codesys 3.0

hm	11. mar. 2009	rev 1.2
	real constants updated to new systax using dot																																																																																																																																																																																																																																																																																																																																																																																																																																																																																																																																																																																																																																																																																																																																																																																																																																																																																																																																																																																																																																																											

*)
          
END_FUNCTION_BLOCK

FUNCTION_BLOCK TUNE2
  VAR_INPUT
    SET : BOOL;
    SU : BOOL;
    SD : BOOL;
    FU : BOOL;
    FD : BOOL;
    RST : BOOL;
    {attribute 'input_constant'}
    SS : REAL := 0.1;
    {attribute 'input_constant'}
    FS : REAL := 5;
    {attribute 'input_constant'}
    Limit_L : REAL;
    {attribute 'input_constant'}
    LIMIT_H : REAL := 100;
    {attribute 'input_constant'}
    RST_val : REAL;
    {attribute 'input_constant'}
    SET_val : REAL := 100;
    {attribute 'input_constant'}
    TR : TIME := TIME#500ms;
    {attribute 'input_constant'}
    S1 : REAL := 2;
    {attribute 'input_constant'}
    S2 : REAL := 10;
  END_VAR
  VAR_OUTPUT
    Y : REAL;
  END_VAR
  VAR
    tx : DWORD;
    start : DWORD;
    state : INT;
    in : BOOL;
    step : REAL;
    SPEED : REAL;
    Y_start : REAL;
  END_VAR

            (* read system time *)
tx := T_PLC_MS();

IF rst THEN
	Y := RST_val;
	state := 0;
ELSIF set THEN
	Y := SET_val;
	state := 0;
ELSIF state > 0 THEN
	(* key has been pushed state machine operating *)
	(* first read the correct input *)
	CASE state OF
		1 :	(* slow up *)
			in := su;
		2 :	(* slow down *)
			in := sd;
		3 :	(* fast up *)
			in := fu;
		4 :	(* fast down *)
			in := fd;
	END_CASE;
	(* check for single step operation *)
	IF NOT in AND tx - start <= TIME_TO_DWORD(TR) THEN
		Y := Y_start + step;
		state := 0;
	(* check if ramp needs to be generated *)
	ELSIF in AND tx - start >= TIME_TO_DWORD(TR) THEN
		Y := Y_start + DWORD_TO_REAL(tx - start - TIME_TO_DWORD(TR)) * speed;
	ELSIF NOT in THEN
		state := 0;
	END_IF;
ELSIF su THEN
	(* slow step up *)
	state := 1;
	start := tx;
	step := ss;
	speed := s1 * 1.0E-3;
	Y_start := Y;
ELSIF sd THEN
	(* slow step down *)
	state := 2;
	start := tx;
	step := -ss;
	speed := -s1 * 1.0E-3;
	Y_start := Y;
ELSIF fu THEN
	(* fast step up *)
	state := 3;
	start := tx;
	step := fs;
	speed := s2 * 1.0E-3;
	y_start := Y;
ELSIF fd THEN
	(* fast step down *)
	state := 4;
	start := tx;
	step := -fs;
	speed := -s2 * 1.0E-3;
	y_start := Y;
END_IF;

(* make sure output does not exceed limits *)
Y := LIMIT(LIMIT_L, Y, LIMIT_H);

(* revision history
hm	3.11.2007		rev 1.0
	original version

hm	16. 3. 2008	rev 1.1
	added type conversions to avoid warnings in codesys 3.0
	improved performance

hm	11. mar. 2009	rev 1.2
	real constants updated to new systax using dot																																																																																																																																																																																																																																																																																																																																																																																																																																																																																																																																																																																																																																																																																																																																																																																																																																																																																																																																																																																																																																																											

*)
          
END_FUNCTION_BLOCK

FUNCTION BAND_B : BYTE
  VAR_INPUT
    X : BYTE;
    B : BYTE;
  END_VAR

            IF X < B THEN
	BAND_B := 0;
ELSIF X > BYTE#255-B THEN
	BAND_B := 255;
ELSE
	BAND_B := X;
END_IF;



(* revision history
hm	21. nov. 2008	rev 1.0
	original version

*)

          
END_FUNCTION

FUNCTION_BLOCK CONTROL_SET1
  VAR_INPUT
    Kt : REAL;
    Tt : REAL;
    PI : BOOL;
    PID : BOOL;
    {attribute 'input_constant'}
    P_K : REAL := 0.5;
    {attribute 'input_constant'}
    PI_K : REAL := 0.45;
    {attribute 'input_constant'}
    PI_TN : REAL := 0.83;
    {attribute 'input_constant'}
    PID_K : REAL := 0.6;
    {attribute 'input_constant'}
    PID_TN : REAL := 0.5;
    {attribute 'input_constant'}
    PID_TV : REAL := 0.125;
  END_VAR
  VAR_OUTPUT
    KP : REAL;
    TN : REAL;
    TV : REAL;
    KI : REAL;
    KD : REAL;
  END_VAR

            IF pi AND PID THEN
	KP := 0.0;
	TN := 0.0;
	TV := 0.0;
ELSIF PID THEN
	KP := PID_K * Kt;
	TN := PID_TN * Tt;
	TV := PID_TV * Tt;
ELSIF PI THEN
	KP := PI_K * Kt;
	TN := PI_TN * Tt;
ELSE
	KP := P_K * Kt;
END_IF;

(* KI and KD are calculated *)
IF tn > 0.0 THEN KI := KP / TN; ELSE KI := 0.0; END_IF;
KD := KP * TV;

(* revision history
hm	4. nov 2007	rev 1.0
	original version

hm	11. mar. 2009	rev 1.1
	real constants updated to new systax using dot																																																																																																																																																																																																																																																																																																																																																																																																																																																																																																																																																																																																																																																																																																																																																																																																																																																																																																																																																																																																																																																											

*)
          
END_FUNCTION_BLOCK

FUNCTION_BLOCK CONTROL_SET2
  VAR_INPUT
    KS : REAL;
    TU : REAL;
    TG : REAL;
    PI : BOOL;
    PID : BOOL;
    {attribute 'input_constant'}
    P_K : REAL := 1;
    {attribute 'input_constant'}
    PI_K : REAL := 0.9;
    {attribute 'input_constant'}
    PI_TN : REAL := 3.33;
    {attribute 'input_constant'}
    PID_K : REAL := 1.2;
    {attribute 'input_constant'}
    PID_TN : REAL := 2;
    {attribute 'input_constant'}
    PID_TV : REAL := 0.5;
  END_VAR
  VAR_OUTPUT
    KP : REAL;
    TN : REAL;
    TV : REAL;
    KI : REAL;
    KD : REAL;
  END_VAR
  VAR
    TX : REAL;
  END_VAR

            IF TU > 0.0 AND KS > 0.0 THEN TX := TG / TU / KS; END_IF;
IF pi AND PID THEN
	KP := 0.0;
	TN := 0.0;
	TV := 0.0;
ELSIF PID THEN
	KP := PID_K * TX;
	TN := PID_TN * TU;
	TV := PID_TV * TU;
ELSIF PI THEN
	KP := PI_K * TX;
	TN := PI_TN * TU;
ELSE
	KP := P_K * TX;
END_IF;

(* KI and KD are calculated *)
IF TN > 0.0 THEN KI := KP / TN; ELSE KI := 0.0; END_IF;
KD := KP * TV;

(* revision history
hm	4. nov 2007	rev 1.0
	original version

hm	11. mar. 2009	rev 1.1
	real constants updated to new systax using dot																																																																																																																																																																																																																																																																																																																																																																																																																																																																																																																																																																																																																																																																																																																																																																																																																																																																																																																																																																																																																																																											

*)
          
END_FUNCTION_BLOCK

FUNCTION CTRL_IN : REAL
  VAR_INPUT
    SET_POINT : REAL;
    ACTUAL : REAL;
    NOISE : REAL;
  END_VAR

            (* calculate the process error DIFF *)
CTRL_IN := DEAD_ZONE(SET_POINT - ACTUAL, NOISE);


(* revision history
hm 	2. jun. 2008 	rev 1.0
	original version

*)
          
END_FUNCTION

FUNCTION_BLOCK CTRL_OUT
  VAR_INPUT
    CI : REAL;
    OFFSET : REAL;
    MAN_IN : REAL;
    LIM_L : REAL;
    LIM_H : REAL;
    MANUAL : BOOL;
  END_VAR
  VAR_OUTPUT
    Y : REAL;
    LIM : BOOL;
  END_VAR

            Y := SEL(MANUAL, CI, MAN_IN) + OFFSET;

(* Limit the output *)
IF Y > LIM_L AND Y < LIM_H THEN
	LIM := FALSE;
ELSE
	Y := LIMIT(LIM_L, Y, LIM_H);
	LIM := TRUE;
END_IF;



(* revision history
hm 	2. jun. 2008 	rev 1.0
	original version

hm	5. nov. 2008	rev 1.1
	optimized code
*)
          
END_FUNCTION_BLOCK

FUNCTION_BLOCK CTRL_PI
  VAR_INPUT
    ACT : REAL;
    SET : REAL;
    SUP : REAL;
    OFS : REAL;
    M_I : REAL;
    MAN : BOOL;
    RST : BOOL;
    KP : REAL := 1;
    KI : REAL := 1;
    LL : REAL := -1000;
    LH : REAL := 1000;
  END_VAR
  VAR_OUTPUT
    Y : REAL;
    DIFF : REAL;
    LIM : BOOL;
  END_VAR
  VAR
    pi : FT_PIWL;
    co : CTRL_OUT;
  END_VAR

            DIFF := CTRL_IN(SET, ACT, SUP);
pi(in := DIFF, kp := KP, ki := KI, lim_l := LL, lim_h := LH, rst := RST);
co(ci := pi.Y, OFFSET := OFS, man_in := M_I, lim_l := LL, lim_h := LH, MANUAL := MAN);
Y := co.Y;
LIM := co.LIM;


(* revision history
hm 	31.10.2007 		rev 1.0
	original version

hm	3.11.2007		rev 1.1
	added noise input to filter noise
	added output diff
	set limit output false when output is within limits
	overfolw was not set correctly

hm	5. jan 2008		rev 1.2
	improved performance

hm	20. jun. 2008	rev 2.0
	rewritten using new modular approach

*)
          
END_FUNCTION_BLOCK

FUNCTION_BLOCK CTRL_PID
  VAR_INPUT
    ACT : REAL;
    SET : REAL;
    SUP : REAL;
    OFS : REAL;
    M_I : REAL;
    MAN : BOOL;
    RST : BOOL;
    KP : REAL := 1;
    TN : REAL := 1;
    TV : REAL := 1;
    LL : REAL := -1000;
    LH : REAL := 1000;
  END_VAR
  VAR_OUTPUT
    Y : REAL;
    DIFF : REAL;
    LIM : BOOL;
  END_VAR
  VAR
    pid : FT_PIDWL;
    co : CTRL_OUT;
  END_VAR

            DIFF := CTRL_IN(SET, ACT, SUP);
pid(in := DIFF, kp := KP, tn := TN, tv := TV, lim_l := LL, lim_h := LH, rst := RST);
co(ci := pid.Y, OFFSET := OFS, man_in := M_I, lim_l := LL, lim_h := LH, MANUAL := MAN);
Y := co.Y;
LIM := co.LIM;



(* revision history

hm 1.12.2006	 	rev 1.1
	changed algorithm to trapezregel for higher accuracy.

hm 3.1.2007		rev 1.2
	added integ_band to select when the integrator is active.

hm	3.3.2007		rev 1.3
	added default values to inputs KP, TN, TV, LIMIT_L und LIMIT_H.

hm 31.oct 2007	rev 1.4
	total rewrite of the module to avoid failures when one of the limits is 0

hm	3.11.2007	rev 1.5
	added noise input to filter noise
	added output diff
	set limit output false when output is within limits
	overfolw was not set correctly

hm	5. jan 2008	rev 1.6
	improved code for better performance
*)
          
END_FUNCTION_BLOCK

FUNCTION_BLOCK CTRL_PWM
  VAR_INPUT
    CI : REAL;
    MAN_IN : REAL;
    MANUAL : BOOL;
    F : REAL;
  END_VAR
  VAR_OUTPUT
    Q : BOOL;
  END_VAR
  VAR
    PW : PWM_DC;
  END_VAR

            PW(F := F, DC := SEL(MANUAL,CI,MAN_IN));
Q := PW.Q;


(* revision history
hm 3. jun. 2008 	rev 1.0
	original version

hm	21. oct. 2008	rev 1.1
	optimized code

*)
          
END_FUNCTION_BLOCK

FUNCTION DEAD_BAND : REAL
  VAR_INPUT
    X : REAL;
    L : REAL;
  END_VAR

            IF X > L THEN
	DEAD_BAND := X - L;
ELSIF X < -L THEN
	DEAD_BAND := X + L;
ELSE
	DEAD_BAND := 0.0;
END_IF;


(* revision history
hm	2. nov. 2007	rev 1.0
	original version

hm	14. jun. 2008	rev 1.1
	improved performance

hm	18. jan. 2011	rev 1.2
	assign 0 before return
*)
          
END_FUNCTION

FUNCTION_BLOCK DEAD_BAND_A
  VAR_INPUT
    X : REAL;
    T : TIME;
    KL : REAL := 1;
    LM : REAL;
  END_VAR
  VAR_OUTPUT
    Y : REAL;
    L : REAL;
  END_VAR
  VAR
    tp1 : FT_PT1;
    tp2 : FT_PT1;
  END_VAR

            (* filter the input signal *)
tp1(in := X, T:= T);

(* filter the HF portion to generate a stable L *)
tp2(in := ABS(tp1.out - X), T := MULTIME(T, 4.0));

(* now we determine L which is half the width of the dead band *)
L := MIN(KL * tp2.out, LM);

IF X > L THEN
	Y := X - L;
ELSIF X < -L THEN
	Y := X + L;
ELSE
	Y := 0.0;
END_IF;


(* revision history
hm	14. jun. 2008	rev 1.0
	original version

hm	11. mar. 2009	rev 1.1
	real constants updated to new systax using dot

*)
          
END_FUNCTION_BLOCK

FUNCTION DEAD_ZONE : REAL
  VAR_INPUT
    X : REAL;
    L : REAL;
  END_VAR

            IF ABS(x) > L THEN
	dead_zone := X;
ELSE
	DEAD_ZONE := 0.0;
END_IF;

(* revision history
hm	12. feb. 2007	rev 1.0
	original version

hm	14. jun. 2008	rev 1.1
	improved performance

hm	11. mar. 2009	rev 1.2
	real constants updated to new systax using dot

*)
          
END_FUNCTION

FUNCTION_BLOCK DEAD_ZONE2
  VAR_INPUT
    X : REAL;
    L : REAL;
  END_VAR
  VAR_OUTPUT
    Y : REAL;
  END_VAR

            IF ABS(x) > L THEN
	Y := X;
ELSIF Y > 0.0 THEN
	Y := L;
ELSE
	Y := -L;
END_IF;



(* revision history

hm	12. feb. 2007	rev 1.0
	original version

hm	11. mar. 2009	rev 1.1
	real constants updated to new systax using dot

*)

          
END_FUNCTION_BLOCK

FUNCTION_BLOCK FT_DERIV
  VAR_INPUT
    in : REAL;
    K : REAL := 1;
    run : BOOL := TRUE;
  END_VAR
  VAR_OUTPUT
    out : REAL;
  END_VAR
  VAR
    old : REAL;
    tx : DWORD;
    last : DWORD;
    init : BOOL;
    tc : REAL;
  END_VAR

            (* read system time *)
tx := T_PLC_US();
tc := DWORD_TO_REAL(tx - last);
last := tx;

(* init on first startup *)
IF NOT init THEN
	init := TRUE;
	old := in;
ELSIF run AND tc > 0.0 THEN
	out := (in - old) / tc * 1000000.0 * K;
	old := in;
ELSE
	out := 0.0;
END_IF;



(*
hm 3.1.2007			rev 1.1
	added init code for startup
	set the default for K to 1

hm	15. sep 2007	rev 1.2
	replaced Time() with T_PLC_US for compatibility and performance reasons
	increased accuracy and work in microseconds internally

hm 29 oct 2007	rev 1.3
	prohibit calculation when tx - last = 0 to avoid division by 0 and increase accuracy on fast systems

hm	6. nov. 2008	rev 1.4
	improved performance

hm	11. mar. 2009	rev 1.5
	inproved code
*)
          
END_FUNCTION_BLOCK

FUNCTION_BLOCK FT_IMP
  VAR_INPUT
    in : REAL;
    T : TIME;
    K : REAL := 1;
  END_VAR
  VAR_OUTPUT
    out : REAL;
  END_VAR
  VAR
    t1 : FT_PT1;
  END_VAR

            T1(in:= in, T:=T);
out := (in - t1.out) * K;

(*
hm 3.1.2007	rev 1.1
	added factor K

*)
          
END_FUNCTION_BLOCK

FUNCTION_BLOCK FT_INT
  VAR_INPUT
    IN : REAL;
    K : REAL := 1;
    RUN : BOOL := TRUE;
    RST : BOOL;
    OUT_MIN : REAL := -1E+37;
    OUT_MAX : REAL := 1E+37;
  END_VAR
  VAR_OUTPUT
    OUT : REAL;
    LIM : BOOL;
  END_VAR
  VAR
    INTeg : INTEGRATE;
  END_VAR

            IF rst THEN
	out := 0.0;
ELSE
	integ(X := IN, E := RUN, K := K, Y := out);
END_IF;

(* limit the outputs *)
IF out >= OUT_MAX THEN
	out := out_max;
	LIM := TRUE;
ELSIF out <= out_min THEN
	out := out_min;
	lim := TRUE;
ELSE
	lim := FALSE;
END_IF;


(*
hm 13.12.2006	rev 1.1
	changed to "trapezregel" which increases accuracy
	before out := out + in * time new: out := out + (in + in_last) / 2 * time

hm 15.1.2007		rev 1.2
	added default for k to be 1.

hm	15.9.2007		rev 1.3
	replaced time() with T_PLC_US for compatibility and performance reason
	increased internal accuracy to microseconds

hm 29. oct 2007		rev 1.4
	changed code so int will not be called is time difference is 0 to increase accuracy on systems
	with cycle times below 1ms

hm	2. dec 2007	 	rev 1.5
	changed code for better performance

hm	5. jan 2008		rev 1.6
	further improvements in performance

hm	8. feb 2008		rev 1.7
	deleted limits +/- 1000 now limit is the range of real
	added variables out1 and out2 to extend the resolution
	corrected an error with elapsed time
	deleted unusfull output ET

hm	13. mar 2008	rev 1.8
	changed preset value out_min to -1e37.
	stop integrator at the limits.

hm	16. mar 2008	rev 1.9
	added type conversion to avoid warning under codesys 3.0

hm	2. jun. 2008	rev 2.0
	rewritten with clear code
	limits can now be set without run

hm	3. nov. 2008	rev 2.1
	optimized code using INTEGRATE and LIMX

hm	10. mar. 2009	rev 2.2
	removed nested comments
*)

          
END_FUNCTION_BLOCK

FUNCTION_BLOCK FT_INT2
  VAR_INPUT
    IN : REAL;
    K : REAL := 1;
    RUN : BOOL := TRUE;
    RST : BOOL;
    OUT_MIN : REAL := -1E+38;
    OUT_MAX : REAL := 1E+38;
  END_VAR
  VAR_OUTPUT
    OUT : REAL;
    LIM : BOOL;
  END_VAR
  VAR
    integ : INTEGRATE;
    ix : REAL;
    val : REAL2;
  END_VAR

            IF RST THEN
	val := R2_SET(0.0);
	out := 0.0;
ELSE
	integ(X := IN, E := RUN, K := K, Y := ix);
	val := R2_ADD(val, ix);
	ix := 0.0;
	OUT := val.RX;
END_IF;

(* check output for limits *)
IF out > OUT_MIN AND out < OUT_MAX THEN
	LIM := FALSE;
ELSE
	OUT := LIMIT(OUT_MIN, OUT, OUT_MAX);
	val := R2_SET(OUT);
	LIM := TRUE;
END_IF;



(*	revision history
hm	2. jun. 2008	rev 1.0
	original version

hm	5. nov. 2008	rev 1.1
	rewritten code using integrate

hm	11. mar. 2009	rev 1.2
	real constants updated to new systax using dot

*)

          
END_FUNCTION_BLOCK

FUNCTION_BLOCK FT_PD
  VAR_INPUT
    IN : REAL;
    KP : REAL := 1;
    TV : REAL := 1;
  END_VAR
  VAR_OUTPUT
    Y : REAL;
  END_VAR
  VAR
    diff : FT_DERIV;
  END_VAR

            (* run differentiator *)
diff(IN := IN, K := TV);

(* combine both values *)
Y := KP * (diff.out + IN);



(* revision history
hm 	3. jun. 2008 	rev 1.0
	original version


*)
          
END_FUNCTION_BLOCK

FUNCTION_BLOCK FT_PDT1
  VAR_INPUT
    IN : REAL;
    KP : REAL := 1;
    TV : REAL := 1;
    T1 : REAL := 1;
  END_VAR
  VAR_OUTPUT
    Y : REAL;
  END_VAR
  VAR
    diff : FT_DERIV;
    TP : FT_PT1;
  END_VAR

            (* run differentiator *)
diff(IN := IN, K := TV);

(* Run PT1 filter *)
tp(in := diff.out, T := REAL_TO_TIME(T1));

(* combine both values *)
Y := KP * (tp.out + IN);



(* revision history
hm 	3. jun. 2008 	rev 1.0
	original version


*)
          
END_FUNCTION_BLOCK

FUNCTION_BLOCK FT_PI
  VAR_INPUT
    IN : REAL;
    KP : REAL := 1;
    KI : REAL := 1;
    ILIM_L : REAL := -1E+38;
    ILIM_H : REAL := 1E+38;
    IEN : BOOL := TRUE;
    RST : BOOL;
  END_VAR
  VAR_OUTPUT
    Y : REAL;
    LIM : BOOL;
  END_VAR
  VAR
    integ : FT_INT;
  END_VAR

            (* run integrator *)
integ(IN := IN, K := KI, RUN := IEN, RST := RST, OUT_MIN := ILIM_L, OUT_MAX := ILIM_H);

(* check if integrator has reached its limits and set overflow *)
LIM := integ.LIM;
Y := KP * IN + integ.Out;



(* revision history
hm 	3. jun. 2008 	rev 2.0
	original version


*)
          
END_FUNCTION_BLOCK

FUNCTION_BLOCK FT_PID
  VAR_INPUT
    IN : REAL;
    KP : REAL := 1;
    TN : REAL := 1;
    TV : REAL := 1;
    ILIM_L : REAL := -1E+38;
    ILIM_H : REAL := 1E+38;
    IEN : BOOL := TRUE;
    RST : BOOL;
  END_VAR
  VAR_OUTPUT
    Y : REAL;
    LIM : BOOL;
  END_VAR
  VAR
    integ : FT_INT;
    diff : FT_DERIV;
  END_VAR

            (* run integrator only if TN > 0 *)
IF TN > 0.0 THEN
	integ(IN := IN, K := 1.0 / TN, RUN := IEN, RST := RST, OUT_MIN := ILIM_L, OUT_MAX := ILIM_H);
ELSE
	integ(RST := FALSE);
END_IF;

(* run differentiator *)
diff(IN := IN, K := TV);

(* combine both values *)
Y := KP * (integ.Out + diff.out + IN);

(* check if integrator has reached its limits and set overflow *)
LIM := integ.LIM;



(* revision history
hm 3. jun. 2008 	rev 2.0
	original version

hm	11. mar. 2009	rev 2.1
	real constants updated to new systax using dot

*)
          
END_FUNCTION_BLOCK

FUNCTION_BLOCK FT_PIDW
  VAR_INPUT
    IN : REAL;
    KP : REAL := 1;
    TN : REAL := 1;
    TV : REAL := 1;
    LIM_L : REAL := -1E+38;
    LIM_H : REAL := 1E+38;
    RST : BOOL;
  END_VAR
  VAR_OUTPUT
    Y : REAL;
    LIM : BOOL;
  END_VAR
  VAR
    integ : INTEGRATE;
    diff : FT_DERIV;
    YI : REAL;
  END_VAR

            (* run the integrator *)
IF tn = 0.0 OR rst THEN
	integ(E := FALSE, Y := YI);
	YI := 0.0;
ELSE
	integ(X := IN, K := 1.0 / TN, E := NOT LIM, Y := YI);
END_IF;

(* add up integrator and linear part *)
Y := KP * (IN + YI);

(* run differentiator *)
diff(IN := IN, K := TV);

(* set lim before differentiator is added to stop integrator if necessary *)
IF Y > LIM_L AND Y < LIM_H THEN
	LIM := FALSE;
ELSE
	LIM := TRUE;
END_IF;

(* add differential part and limit output Y *)

Y := LIMIT(LIM_L, Y + KP * diff.out, LIM_H);




(* revision history
hm 3. jun. 2008 	rev 1.0
	original version

hm	5. nov. 2008	rev 1.1
	changed code to use integrate

hm	11. mar. 2009	rev 1.2
	real constants updated to new systax using dot

*)
          
END_FUNCTION_BLOCK

FUNCTION_BLOCK FT_PIDWL
  VAR_INPUT
    IN : REAL;
    KP : REAL := 1;
    TN : REAL := 1;
    TV : REAL := 1;
    LIM_L : REAL := -1E+38;
    LIM_H : REAL := 1E+38;
    RST : BOOL;
  END_VAR
  VAR_OUTPUT
    Y : REAL;
    LIM : BOOL;
  END_VAR
  VAR
    piwl : FT_PIWL;
    diff : FT_DERIV;
  END_VAR

            (* if rst then *)
IF rst THEN
	piwl(rst := TRUE);
	piwl.RST := FALSE;
ELSE
	(* run PIWL controller first *)
	(* we need to check if TN = 0 and do alternative calls *)
	IF TN = 0.0 THEN
		piwl(in := IN * KP, KP := 1.0, KI := 0.0, LIM_L := LIM_L, LIM_H := LIM_H);
	ELSE
		piwl(in := IN * KP, KP := 1.0, KI := 1.0 / TN, LIM_L := LIM_L, LIM_H := LIM_H);
	END_IF;

	(* run differentiator and add_to_output *)
	diff(IN := IN, K := KP * TV);
	Y := piwl.Y + diff.out;

	(* limit the output *)
	IF Y < LIM_L THEN
		LIM := TRUE;
		Y := LIM_L;
	ELSIF Y > LIM_H THEN
		LIM := TRUE;
		Y := LIM_H;
	ELSE
		LIM := FALSE;
	END_IF;
END_IF;



(* revision history
hm 13. jun. 2008 	rev 1.0
	original version

hm	25. jan 2008	rev 1.1
	multiply differential part with KP

hm	11. mar. 2009	rev 1.2
	real constants updated to new systax using dot

hm	13. nov. 2009	rev 1.3
	fixed code for negative KP

*)
          
END_FUNCTION_BLOCK

FUNCTION_BLOCK FT_PIW
  VAR_INPUT
    IN : REAL;
    KP : REAL := 1;
    KI : REAL := 1;
    LIM_L : REAL := -1E+38;
    LIM_H : REAL := 1E+38;
    RST : BOOL;
  END_VAR
  VAR_OUTPUT
    Y : REAL;
    LIM : BOOL;
  END_VAR
  VAR
    integ : FT_INT;
  END_VAR

            (* run integrator *)
integ(IN := IN, K := KI, RUN := NOT LIM, RST := RST);

(* set output value *)
Y := KP * IN + integ.Out;

(* check for limits and set integrator for anti wind up *)
IF Y < LIM_L THEN
	Y := LIM_L;
	LIM := TRUE;
ELSIF Y > LIM_H THEN
	Y := LIM_H;
	LIM := TRUE;
ELSE
	LIM := FALSE;
END_IF;



(* revision history
hm 	3. jun. 2008 	rev 1.0
	original version


*)
          
END_FUNCTION_BLOCK

FUNCTION_BLOCK FT_PIWL
  VAR_INPUT
    IN : REAL;
    KP : REAL := 1;
    KI : REAL := 1;
    LIM_L : REAL := -1E+38;
    LIM_H : REAL := 1E+38;
    RST : BOOL;
  END_VAR
  VAR_OUTPUT
    Y : REAL;
    LIM : BOOL;
  END_VAR
  VAR
    init : BOOL;
    tx : DWORD;
    tc : REAL;
    t_last : DWORD;
    in_last : REAL;
    i : REAL;
    p : REAL;
  END_VAR

            (* initialize at power_up *)
IF NOT init OR RST THEN
	init := TRUE;
	in_last := in;
	t_last := T_PLC_US();
	i := 0.0;
	tc := 0.0;
ELSE
	(* read last cycle time in Microseconds *)
	tx := T_PLC_US();
	tc := DWORD_TO_REAL(tx - t_last);
	t_last := tx;

	(* calculate proportional part *)
	p := KP * IN;

	(* run integrator *)
	i := (IN + in_last) * 5.0E-7 * KI * tc + i;
	in_last := IN;

	(* calculate output Y *)
	Y := p + i;

	(* check output for limits *)
	IF Y >= LIM_H THEN
		Y := LIM_H;
		IF ki <> 0.0 THEN
			i := LIM_H - p;
		ELSE
			i := 0.0;
		END_IF;
		LIM := TRUE;
	ELSIF Y <= LIM_L THEN
		Y := LIM_L;
		IF ki <> 0.0 THEN
			i := LIM_L - p;
		ELSE
			i := 0.0;
		END_IF;
		LIM := TRUE;
	ELSE
		LIM := FALSE;
	END_IF;
END_IF;




(* revision history
hm 13. jun. 2008 	rev 1.0
	original version

hm	27. oct. 2008	rev 1.1
	integrator will not be adjusted when ki = 0

hm	25. jan 2009	rev 1.2
	module will also work with negative K

hm	11. mar. 2009	rev 1.3
	real constants updated to new systax using dot

*)
          
END_FUNCTION_BLOCK

FUNCTION_BLOCK FT_PT1
  VAR_INPUT
    in : REAL;
    T : TIME;
    K : REAL := 1;
  END_VAR
  VAR_OUTPUT
    out : REAL;
  END_VAR
  VAR
    last : DWORD;
    tx : DWORD;
    init : BOOL;
  END_VAR

            (* read system time *)
tx := T_PLC_US();

(* startup initialisation *)
IF NOT init OR T = t#0s THEN
	init := TRUE;
	out := K * in;
ELSE
	out := out + (in * K - out) * DWORD_TO_REAL(Tx - last) / TIME_TO_REAL(T) * 1.0E-3;
	IF ABS(out) < 1.0E-20 THEN out := 0.0; END_IF;
END_IF;
last := tx;


(*
hm 1.1.2007	rev 1.1
	corrected error while startup value was not correct
	for very small time values real output would run out of range.

hm 3.1.2007	rev 1.2
	corrected an error for falling edge failures.
	added output faktor K.

hm 27. 2. 2007	rev 1.3
	output will be input during init for definitive startup condition.

hm	15.9.2007	rev 1.4
	changed time() to T_PLC_US() for compatibilitxy resons
	increased internal accuracy to Microseconds instead of Milliseconds

hm	23. oct 2007	rev 1.5
	added out := in to the init statements

hm	30. nov 2007	rev 1.6
	changed out to be K * in during initialization

hm	5. jan 2008	rev 1.7
	improved code for better performance

hm	16. mar. 2008	rev 1.8
	added type conversion to avoid warning under codesys 3.0

hm	14. jun. 2008	rev 1.9
	improved code

hm	11. mar. 2009	rev 1.10
	real constants updated to new systax using dot

hm	18. jan. 2011	rev 1.11
	avoid underrun of out
*)
          
END_FUNCTION_BLOCK

FUNCTION_BLOCK FT_PT2
  VAR_INPUT
    in : REAL;
    T : TIME;
    D : REAL;
    K : REAL := 1;
  END_VAR
  VAR_OUTPUT
    out : REAL;
  END_VAR
  VAR
    init : BOOL;
    int1 : INTEGRATE;
    int2 : INTEGRATE;
    tn : REAL;
    I1 : REAL;
    I2 : REAL;
    tn2 : REAL;
  END_VAR

            (* startup initialisation *)
IF NOT init OR T = T#0s THEN
	init := TRUE;
	out := K * in;
	I2 := out;
ELSE
	TN := TIME_TO_REAL(T) * 1.0E-3;
	tn2 := TN * TN;
	int1(X := in * K / tn2 - I1 * 0.5 * D / TN - I2 / TN2, Y := I1);
	int2(X := I1,Y := I2);
	out := I2;
END_IF;


(* revision history

15.1.2007 hm		rev 1.1
	changed formula to new more acurate formula

hm 15.9.2007		rev 1.2
	deleted unused code for init system time reading tx	

hm	30.11.2007	rev 1.3
	changed out to be K * in during initialization
	avoind divide by 0 if tn = 0

hm	3. nov. 2008	rev 1.4
	optimized code and fixed a problem with init

hm	11. mar. 2009	rev 1.5
	real constants updated to new systax using dot

*)
          
END_FUNCTION_BLOCK

FUNCTION_BLOCK FT_TN16
  VAR_INPUT
    in : REAL;
    T : TIME;
  END_VAR
  VAR_OUTPUT
    out : REAL;
    trig : BOOL;
  END_VAR
  VAR
    length : INT := 16;
    X : ARRAY[0..15] OF REAL;
    cnt : INT;
    last : TIME;
    tx : TIME;
    init : BOOL;
  END_VAR

            (* read system time *)
tx := DWORD_TO_TIME(T_PLC_MS());

trig := FALSE;
IF NOT init THEN
	x[cnt] := in;
	init := TRUE;
	last := tx;
ELSIF tx - last >= T / length THEN
	IF cnt = length - 1 THEN cnt := 0; ELSE cnt := cnt + 1; END_IF;
	Out := X[cnt];
	x[cnt] := in;
	last := tx;
	Trig := TRUE;
END_IF;

(* revision history
hm		1. jan 2007	rev 1.0
	original version

hm		16. sep 2007	rev 1.1
	changes time() to T_plc_ms() for compatibility reasons

*)
          
END_FUNCTION_BLOCK

FUNCTION_BLOCK FT_TN64
  VAR_INPUT
    in : REAL;
    T : TIME;
  END_VAR
  VAR_OUTPUT
    out : REAL;
    trig : BOOL;
  END_VAR
  VAR
    length : INT := 64;
    X : ARRAY[0..63] OF REAL;
    cnt : INT;
    last : TIME;
    tx : TIME;
    init : BOOL;
  END_VAR

            (* read system time *)
tx := DWORD_TO_TIME(T_PLC_MS());

trig := FALSE;
IF NOT init THEN
	x[cnt] := in;
	init := TRUE;
	last := tx;
ELSIF tx - last >= T / length THEN
	IF cnt = length - 1 THEN cnt := 0; ELSE cnt := cnt + 1; END_IF;
	Out := X[cnt];
	x[cnt] := in;
	last := tx;
	trig := TRUE;
END_IF;

(* revision history
hm		1. jan 2007		rev 1.0
	original version

hm		16. sep 2007	rev 1.1
	changes time() to T_plc_ms() for compatibility reasons

*)
          
END_FUNCTION_BLOCK

FUNCTION_BLOCK FT_TN8
  VAR_INPUT
    in : REAL;
    T : TIME;
  END_VAR
  VAR_OUTPUT
    out : REAL;
    trig : BOOL;
  END_VAR
  VAR
    length : INT := 8;
    X : ARRAY[0..7] OF REAL;
    cnt : INT;
    last : TIME;
    tx : TIME;
    init : BOOL;
  END_VAR

            tx := DWORD_TO_TIME(T_PLC_MS());
trig := FALSE;
IF NOT init THEN
	x[cnt] := in;
	init := TRUE;
	last := tx;
ELSIF tx - last >= T / length THEN
	IF cnt = length - 1 THEN cnt := 0; ELSE cnt := cnt + 1; END_IF;
	Out := X[cnt];
	x[cnt] := in;
	last := tx;
	trig := TRUE;
END_IF;

(* revision history
hm		1. jan 2007		rev 1.0
	original version

hm		16. sep 2007	rev 1.1
	changes time() to T_plc_ms() for compatibility reasons

*)
          
END_FUNCTION_BLOCK

FUNCTION_BLOCK HYST
  VAR_INPUT
    In : REAL;
    ON : REAL;
    OFF : REAL;
  END_VAR
  VAR_OUTPUT
    Q : BOOL;
    win : BOOL;
  END_VAR

            IF ON >= OFF THEN
	IF IN < OFF THEN
		Q := FALSE;
		WIN := FALSE;
	ELSIF  IN > ON THEN
		Q := TRUE;
		WIN := FALSE;
	ELSE
		WIN := TRUE;
	END_IF;
ELSE
	IF IN > OFF THEN
		Q := FALSE;
		WIN := FALSE;
	ELSIF  IN < ON THEN
		Q := TRUE;
		WIN := FALSE;
	ELSE
		WIN := TRUE;
	END_IF;
END_IF;


(* revision history
hm		2.  jun 2008	rev 1.0
	original version

*)
          
END_FUNCTION_BLOCK

FUNCTION_BLOCK HYST_1
  VAR_INPUT
    In : REAL;
    high : REAL;
    low : REAL;
  END_VAR
  VAR_OUTPUT
    Q : BOOL;
    win : BOOL;
  END_VAR

            IF in < low THEN
	Q := FALSE;
	win := FALSE;
ELSIF in > high THEN
	Q := TRUE;
	win := FALSE;
ELSE
	win := TRUE;
END_IF;




(* revision history
hm		4.  aug. 2006	rev 1.0
	original version

hm		2. jun. 2008	rev 1.1
	improved performance
*)
          
END_FUNCTION_BLOCK

FUNCTION_BLOCK HYST_2
  VAR_INPUT
    IN : REAL;
    VAL : REAL;
    HYS : REAL;
  END_VAR
  VAR_OUTPUT
    Q : BOOL;
    WIN : BOOL;
  END_VAR
  VAR
    tmp : REAL;
  END_VAR

            tmp := val - hys * 0.5;
IF in < tmp THEN
	Q := FALSE;
	win := FALSE;
ELSIF in > tmp + hys THEN
	Q := TRUE;
	win := FALSE;
ELSE
	win := TRUE;
END_IF;



(* revision history
hm		4. aug 2006	rev 1.0
	original version

hm		5. jan 2008	rev 1.1
	improved code for better performance

hm		2. jun. 2008	rev 1.2
	improved performance
*)
          
END_FUNCTION_BLOCK

FUNCTION_BLOCK HYST_3
  VAR_INPUT
    in : REAL;
    hyst : REAL;
    val1 : REAL;
    val2 : REAL;
  END_VAR
  VAR_OUTPUT
    Q1 : BOOL;
    Q2 : BOOL;
  END_VAR
  VAR
    X : REAL;
  END_VAR

            X := hyst * 0.5;
IF in < val1 - X THEN
	q1 := TRUE;
ELSIF in > val1 + X THEN
	q1 := FALSE;
END_IF;
IF in < val2 - X THEN
	q2 := FALSE;
ELSIF in > val2 + X THEN
	q2 := TRUE;
END_IF;



(* revision history
hm	22. jan 2007	rev 1.0
	original version

hm	27. dec 2007	rev 1.1
	changed code for better performance

hm	5. jan 2008	rev 1.2
	further performance iprovements

*)

          
END_FUNCTION_BLOCK

FUNCTION_BLOCK INTEGRATE
  VAR_INPUT
    E : BOOL := TRUE;
    X : REAL;
    K : REAL := 1;
  END_VAR
  VAR_IN_OUT
    Y : REAL;
  END_VAR
  VAR
    X_last : REAL;
    init : BOOL;
    last : DWORD;
    tx : DWORD;
  END_VAR

            (*read system time *)
tx := T_PLC_MS();

IF NOT init THEN
	init := TRUE;
	X_last := X;
ELSIF E THEN
	Y := (X + X_LAST) * 0.5E-3 * DWORD_TO_REAL(tx-last) * K + Y;
	X_last := X;
END_IF;
last := tx;



(*
hm 3. nov. 2008	rev 1.0
original version
	
*)

          
END_FUNCTION_BLOCK

FUNCTION_BLOCK ASTRO
  VAR_INPUT
    m : REAL;
    AE : REAL;
    PC : REAL;
    LJ : REAL;
  END_VAR
  VAR_OUTPUT
    Ym : REAL;
    YAE : REAL;
    YPC : REAL;
    YLJ : REAL;
  END_VAR

            YAE :=	AE
		+ m * 6.6845871535E-012
		+ PC * 206265.0
		+ LJ * 63240.0;
Ym := YAE * 149.597870E9;
YPC := YAE * 4.8481322570E-006;
YLJ := YAE * 1.5812776724E-005;


(*
Länge Meter m SI-Basiseinheit
Astronomische Einheit* AE 1 AE = 149,597 870 · E9 m
Parsec pc 1 pc = 206265 AE = 30,857 · E15 m
Lichtjahr Lj 1 Lj = 9,460 530 · E15 m = 63240 AE = 0,306 59 pc
Ångström Å 1 Å = El0 m
typograph. Punkt p 1 p = 0,376 065 mm  im Druckereigewerbe
inch** in 1 in = 2,54 · E2 m = 25,4 mm***
foot ft 1 ft = 0,3048 m = 30,48 cm
yard yd 1 yd = 0,9144 m
mile mile 1 mile = 1609,344 m
Internat. Seemeile sm 1 sm = 1852 m
Fathom fm 1 fm = 1,829 m  in der Seeschifffahrt
*)

(* revision history

hm	27. mar. 2007	rev 1.0
	original version

hm	11. mar. 2009	rev 1.1
	improved code

*)

          
END_FUNCTION_BLOCK

FUNCTION BFT_TO_MS : REAL
  VAR_INPUT
    BFT : INT;
  END_VAR

            BFT_TO_MS := EXPT(BFT, 1.5) * 0.836;


(* revision history
hm	12. 6. 2008		rev 1.0
	original version

*)
          
END_FUNCTION

FUNCTION C_TO_F : REAL
  VAR_INPUT
    celsius : REAL;
  END_VAR

            C_TO_F := celsius * 1.8 + 32.0;


(* revision history

hm	4. aug. 2006	rev 1.0
	original version

hm	11. mar. 2009	rev 1.1
	real constants updated to new systax using dot

*)
          
END_FUNCTION

FUNCTION C_TO_K : REAL
  VAR_INPUT
    Celsius : REAL;
  END_VAR

            C_TO_K := Celsius - phys.T0;

(* revision history

hm	4. aug 2006	rev 1.0
	original version

hm	19. aug 2009	rev 1.1
	fixed calculation error

*)

          
END_FUNCTION

FUNCTION DEG_TO_DIR : STRING(3)
  VAR_INPUT
    DEG : INT;
    N : INT;
    L : INT;
  END_VAR
  VAR
    ly : INT;
  END_VAR

            IF L = 0 THEN ly := LANGUAGE.DEFAULT; ELSE ly := MIN(L, LANGUAGE.LMAX); END_IF;
DEG_TO_DIR := LANGUAGE.DIRS[ly, ((SHL(DEG,N-1) + 45) / 90) MOD SHL(INT#2,N)*SHR(INT#8,N)];



(*
DIR := ((SHL(DEG,N-1) + 45) / 90) MOD SHL(INT#2,N);
explanation :
DIR is calculated BY the following formula:
DIR := ((DIR + 45) / 90) MOD 4 if N = 1 digit
North = 0, East = 1 ....
DIR := ((DIR + 22,5) / 45) MOD 8 if N = 2 digit
convert to integer calculation
DIR := ((DIR*2 + 45) / 90) MOD 8
N = 0, NE = 1 ....
ther above formula replaces 2^N with shift for performance
*)



(* revision histroy
hm	11. jun. 2008	rev 1.0
	original release

hm	22. oct. 2008	rev 1.1
	changed size of string variables to 30
*)
          
END_FUNCTION

FUNCTION DIR_TO_DEG : INT
  VAR_INPUT
    DIR : STRING(3);
    L : INT;
  END_VAR
  VAR
    ly : INT;
    i : INT;
  END_VAR

            IF L = 0 THEN ly := LANGUAGE.DEFAULT; ELSE ly := MIN(L, LANGUAGE.LMAX); END_IF;
FOR i := 0 TO 15 DO
	IF language.DIRS[ly, i] = DIR THEN EXIT; END_IF;
END_FOR;
DIR_TO_DEG := SHR(i * 45 + 1, 1);






(* revision histroy
hm	22. oct. 2008	rev 1.1
	original release

*)
          
END_FUNCTION

FUNCTION_BLOCK ENERGY
  VAR_INPUT
    J : REAL;
    C : REAL;
    Wh : REAL;
  END_VAR
  VAR_OUTPUT
    YJ : REAL;
    YC : REAL;
    YWh : REAL;
  END_VAR

            YJ := J + Wh * 3600.0 + C * 4.1868;
YC := YJ * 0.238845896627496;
YWh := YJ * 2.7777777778E-004;

(*
Arbeit, Energie, Joule* J 1 J = 1 N · m = 1 W · s = (1/3,6) E6 kW · h = 1 kg · m2/s2
Wärmemenge Kilowattstunde kW · h 1 kW · h = 3,6 MJ = 860 kcal
Elektronvolt eV 1 eV = 160,218 92 E21 J
Erg erg 1 erg = 1E7 J
Kalorie calorie 1 calalorie = 4,1868 J = 1,163 E3 W · h
Therm therm 1 therm = 105,50 · 106 J
*)

(* revision history

hm	27. mar. 2007	rev 1.0
	original version

hm	11. mar. 2009	rev 1.1
	improved code

hm 16. jan 2010	rev 1.2
	avoid the string cal in comments for codesys import bug


*)
          
END_FUNCTION_BLOCK

FUNCTION F_TO_C : REAL
  VAR_INPUT
    fahrenheit : REAL;
  END_VAR

            F_TO_C := (fahrenheit - 32.0) * 0.5555555555555;

(* revision history
hm	4. aug 2006	rev 1.0
	original version

hm	11. mar. 2009	rev 1.1
	real constants updated to new systax using dot

*)
          
END_FUNCTION

FUNCTION F_TO_OM : REAL
  VAR_INPUT
    F : REAL;
  END_VAR

            F_TO_OM := math.PI2 * F;


(* revision history
hm	22. jan. 2007	rev 1.0
	original version

hm	18. oct. 2008	rev 1.1
	unsing math constants

*)
          
END_FUNCTION

FUNCTION F_TO_PT : TIME
  VAR_INPUT
    F : REAL;
  END_VAR

            F_TO_PT := DWORD_TO_TIME(REAL_TO_DWORD(1.0 / F * 1000.0));


(* revision history

hm	4. aug. 2006	rev 1.0
	original version

hm	11. mar. 2009	rev 1.1
	real constants updated to new systax using dot

*)

          
END_FUNCTION

FUNCTION GEO_TO_DEG : REAL
  VAR_INPUT
    D : INT;
    M : INT;
    SEC : REAL;
  END_VAR

            GEO_TO_DEG := INT_TO_REAL(D) + INT_TO_REAL(M) * 0.016666666666667 + sec * 0.00027777777777778;


(* revision histroy
hm	22. jan. 2009	rev 1.0
	original release


*)
          
END_FUNCTION

FUNCTION K_TO_C : REAL
  VAR_INPUT
    Kelvin : REAL;
  END_VAR

            K_TO_C := Kelvin + phys.T0;


(* revision history

hm	4. aug 2006	rev 1.0
	original version

hm	19. aug 2009	rev 1.1
	fixed calculation error

*)

          
END_FUNCTION

FUNCTION KMH_TO_MS : REAL
  VAR_INPUT
    kmh : REAL;
  END_VAR

            KMH_TO_MS := kmh * 0.2777777777777;

(* revision history
hm	4. feb 2007		rev 1.0
	original version

hm	6. jan 2008		rev 1.1
	improved performance

*)


          
END_FUNCTION

FUNCTION_BLOCK LENGTH
  VAR_INPUT
    m : REAL;
    p : REAL;
    in : REAL;
    ft : REAL;
    yd : REAL;
    mile : REAL;
    sm : REAL;
    fm : REAL;
  END_VAR
  VAR_OUTPUT
    Ym : REAL;
    Yp : REAL;
    Yin : REAL;
    Yft : REAL;
    Yyd : REAL;
    Ymile : REAL;
    Ysm : REAL;
    Yfm : REAL;
  END_VAR

            Ym :=	m
		+ p * 0.000376065
		+ in * 0.0254
		+ ft * 0.3048
		+ yd * 0.9144
		+ mile * 1609.344
		+ sm * 1852.0
		+ fm * 1.829;
Yp := Ym * 2659.11478068951;
Yin := Ym * 39.37007874016;
Yft := Ym * 3.28083989501;
Yyd := Ym * 1.09361329834;
Ymile := Ym * 0.00062137119;
Ysm := Ym * 0.00053995680;
Yfm := Ym * 0.54674685621;

(*
Länge Meter m SI-Basiseinheit
Astronomische Einheit* AE 1 AE = 149,597 870 · E9 m
Parsec pc 1 pc = 206265 AE = 30,857 · E15 m
Lichtjahr Lj 1 Lj = 9,460 530 · E15 m = 63240 AE = 0,306 59 pc
Ångström Å 1 Å = El0 m
typograph. Punkt p 1 p = 0,376 065 mm  im Druckereigewerbe
inch** in 1 in = 2,54 · E2 m = 25,4 mm***
foot ft 1 ft = 0,3048 m = 30,48 cm
yard yd 1 yd = 0,9144 m
mile mile 1 mile = 1609,344 m
Internat. Seemeile sm 1 sm = 1852 m
Fathom fm 1 fm = 1,829 m  in der Seeschifffahrt
*)

(* revision history

hm	27. mar. 2007	rev 1.0
	original version

hm	11. mar. 2009	rev 1.1
	improved code

*)

          
END_FUNCTION_BLOCK

FUNCTION MS_TO_BFT : INT
  VAR_INPUT
    MS : REAL;
  END_VAR

            MS_TO_BFT := REAL_TO_INT(EXPT(MS * 1.196172, 0.666667));


(* revision history
hm	12. 6. 2008		rev 1.0
	original version

*)
          
END_FUNCTION

FUNCTION MS_TO_KMH : REAL
  VAR_INPUT
    ms : REAL;
  END_VAR

            MS_TO_KMH := ms * 3.6;


          
END_FUNCTION

FUNCTION OM_TO_F : REAL
  VAR_INPUT
    OM : REAL;
  END_VAR

            OM_TO_F := OM / math.PI2;


(* revision history
hm	22. jan. 2007	rev 1.0
	original version

hm	18. oct. 2008	rev 1.1
	using math constants

*)
          
END_FUNCTION

FUNCTION_BLOCK PRESSURE
  VAR_INPUT
    mws : REAL;
    torr : REAL;
    att : REAL;
    atm : REAL;
    pa : REAL;
    bar : REAL;
  END_VAR
  VAR_OUTPUT
    Ymws : REAL;
    Ytorr : REAL;
    Yatt : REAL;
    Yatm : REAL;
    Ypa : REAL;
    Ybar : REAL;
  END_VAR

            Ybar := bar +
		pa * 1.0E-5 +
		0.980665 * att +
		1.01325 * atm +
		0.001333224 * torr +
		0.0980665 * mws;
Ymws := ybar * 10.1971621297793;
Ytorr := ybar * 750.0615050434140;
Yatt := ybar * 1.0197162129779;
yatm := ybar * 0.9869232667160;
Ypa := ybar * 100000.0;


(*
Druck, Pascal Pa 1 Pa = 1 N/m2 = 1 kg/(s2 E m) . 0,75 E 10.2 mmHg
mechanische 1 MPa = 1 N/mm2 . fur Festigkeitsangaben
Spannung Bar bar 1 bar = 105 Pa = 103 mbar = 105 kg/(s2 E m)
Millimeter- mmHg 1 mmHg = 133,322 Pa = 1,333 22 mbar
Quecksilbersaule . nur in Heilkunde zulassig
physik. Atmosphare atm 1 atm = 1,013 25 bar
techn. Atmosphare at 1 at = 1 kp/cm2 = 0,980665 bar
Torr Torr 1 Torr = (101325/760) Pa = 1,333224 mbar
Meter-Wassersaule mWS 1 mWS = 9806,65 Pa = 98,0665 mbar
psi lbf/in2 1 lbf/in2 = 68,947 57 mbar = 6894,757 Pa

*)

(* revision history

hm	27. mar. 2007	rev 1.0
	original version

hm	11. mar. 2009	rev 1.1
	improved code

*)
          
END_FUNCTION_BLOCK

FUNCTION PT_TO_F : REAL
  VAR_INPUT
    PT : TIME;
  END_VAR

            PT_TO_F := 1000.0 / DWORD_TO_REAL(TIME_TO_DWORD(PT));


(*	revision history
hm	4. aug. 2006	rev 1.0
	original version

hm	11. mar. 2009	rev 1.1
	real constants updated to new systax using dot

*)

          
END_FUNCTION

FUNCTION_BLOCK SPEED
  VAR_INPUT
    ms : REAL;
    kmh : REAL;
    kn : REAL;
    mh : REAL;
  END_VAR
  VAR_OUTPUT
    Yms : REAL;
    Ykmh : REAL;
    Ykn : REAL;
    Ymh : REAL;
  END_VAR

            Yms := ms +
		kmh * 0.27777777777778 +
		kn * 0.5144444 +
		mh * 0.44704;
Ykmh := Yms * 3.6;
Ykn := Yms * 1.94384466037535;
Ymh := Yms * 2.23693629205440;

(*
Geschwindigkeit Meter durch Sekunde m/s 1 m/s = 3,6 km/h
km durch (pro) Stunde, nicht Stundenkilometer verwenden
Knoten kn 1 kn = 1 sm/h = 0,5144 m/s

*)

(* revision history
hm	27. mar. 2009	rev 1.0
	original version

hm	11. mar. 2009	rev 1.1
	improved code

*)
          
END_FUNCTION_BLOCK

FUNCTION_BLOCK TEMPERATURE
  VAR_INPUT
    K : REAL;
    C : REAL := -273.15;
    F : REAL := -459.67;
    Re : REAL := -218.52;
    Ra : REAL;
  END_VAR
  VAR_OUTPUT
    YK : REAL;
    YC : REAL;
    YF : REAL;
    YRe : REAL;
    YRa : REAL;
  END_VAR

            YK := K + (C + 273.15) + (F + 459.67) * 0.555555555555 + (Re * 1.25 + 273.15) + (Ra * 0.555555555555);
YC := YK -273.15;
YF := YK * 1.8 - 459.67;
YRe := (YK - 273.15) * 0.8;
YRa := YK * 1.8;


(* revision history
hm	21. feb. 2008	rev 1.0
	original version

*)
          
END_FUNCTION_BLOCK

FUNCTION_BLOCK ALARM_2
  VAR_INPUT
    X : REAL;
    LO_1 : REAL;
    HI_1 : REAL;
    LO_2 : REAL;
    HI_2 : REAL;
    HYS : REAL;
  END_VAR
  VAR_OUTPUT
    Q1_LO : BOOL;
    Q1_HI : BOOL;
    Q2_LO : BOOL;
    Q2_HI : BOOL;
  END_VAR
  VAR
    tmp : REAL;
  END_VAR

            tmp := X - Hys * 0.5;
IF tmp > LO_1 THEN Q1_LO := FALSE; END_IF;
IF tmp > LO_2 THEN Q2_LO := FALSE; END_IF;
IF tmp > HI_1 THEN Q1_HI := TRUE; END_IF;
IF tmp > HI_2 THEN Q2_HI := TRUE; END_IF;
tmp := tmp + hys;
IF tmp < LO_1 THEN Q1_LO := TRUE; END_IF;
IF tmp < LO_2 THEN Q2_LO := TRUE; END_IF;
IF tmp < HI_1 THEN Q1_HI := FALSE; END_IF;
IF tmp < HI_2 THEN Q2_HI := FALSE; END_IF;



(* revision history
hm	19. may. 2008		rev 1.0
	original version

hm	11. mar. 2009	rev 1.1
	improved code
*)

          
END_FUNCTION_BLOCK

FUNCTION_BLOCK BAR_GRAPH
  VAR_INPUT
    X : REAL;
    rst : BOOL;
    {attribute 'input_constant'}
    trigger_Low : REAL;
    {attribute 'input_constant'}
    trigger_High : REAL;
    {attribute 'input_constant'}
    Alarm_low : BOOL;
    {attribute 'input_constant'}
    Alarm_high : BOOL;
    {attribute 'input_constant'}
    log_scale : BOOL;
  END_VAR
  VAR_OUTPUT
    LOW : BOOL;
    Q1 : BOOL;
    Q2 : BOOL;
    Q3 : BOOL;
    Q4 : BOOL;
    Q5 : BOOL;
    Q6 : BOOL;
    HIGH : BOOL;
    Alarm : BOOL;
    Status : BYTE;
  END_VAR
  VAR
    init : BOOL;
    T1 : REAL;
    T2 : REAL;
    T3 : REAL;
    T4 : REAL;
    T5 : REAL;
    temp : REAL;
  END_VAR

            IF NOT init THEN
	init := TRUE;
	IF log_scale THEN
		temp := EXP(LN(Trigger_high / Trigger_low) * 0.166666666666666666666);
		T1 := trigger_low * temp;
		T2 := T1 * temp;
		T3 := T2 * temp;
		T4 := T3 * temp;
		T5 := T4 * temp;
	ELSE
		temp := (trigger_high - trigger_low) * 0.142857142;
		T1 := trigger_low + temp;
		T2 := T1 + temp;
		T3 := T2 + temp;
		T4 := T3 + temp;
		T5 := T4 + temp;
	END_IF;
END_IF;

(* clear outputs before checking *)
Q1 := FALSE;
Q2 := FALSE;
Q3 := FALSE;
Q4 := FALSE;
Q5 := FALSE;
Q6 := FALSE;
status := 110;

(* low, high and alarm can only be cleared with rst depending on alarm_low and alarm_high *)
IF NOT alarm_low THEN low := FALSE; END_IF;
IF NOT alarm_high THEN high := FALSE; END_IF;
IF rst THEN
	alarm := FALSE;
	low := FALSE;
	high := FALSE;
END_IF;

(* check and set outputs *)
IF X < trigger_low THEN
	Low := TRUE;
	status := 111;
	IF alarm_low THEN
		alarm := TRUE;
		status := 1;
	END_IF;
ELSIF X < T1 THEN
	Q1 := TRUE;
ELSIF x < t2 THEN
	Q2 := TRUE;
ELSIF x < t3 THEN
	Q3 := TRUE;
ELSIF x < T4 THEN
	Q4 := TRUE;
ELSIF x < T5 THEN
	q5 := TRUE;
ELSIF x < trigger_high THEN
	q6 := TRUE;
ELSE
	high := TRUE;
	status := 112;
	IF alarm_high THEN
		alarm := TRUE;
		status := 2;
	END_IF;
END_IF;

(* revision history
hm	22. feb 2007	rev 1.0
	original version

hm	2. dec 2007		rev 1.1
	chaged code for better performance

hm	6. jan 2008		rev 1.2
	further performance improvement

*)
          
END_FUNCTION_BLOCK

FUNCTION_BLOCK CALIBRATE
  VAR_INPUT
    X : REAL;
    CO : BOOL;
    CS : BOOL;
    {attribute 'input_constant'}
    Y_Offset : REAL;
    {attribute 'input_constant'}
    Y_Scale : REAL;
  END_VAR
  VAR_OUTPUT
    Y : REAL;
  END_VAR
  VAR RETAIN
    offset : REAL;
    Scale : REAL := 1;
  END_VAR

            (* check for calibration *)
IF CO THEN
	OFFSET := Y_Offset - X;
ELSIF CS THEN
	SCALE := Y_scale / (X + OFFSET);
END_IF;
(* calculate output *)
Y := (X + OFFSET) * SCALE;


(* revision history
hm 22.2.2007		rev 1.2
	changed VAR RETAIN PERSISTENT to VAR RETAIN for better compatibility
	wago lon contollers do not support persisitent

hm	11. mar. 2009	rev 1.3
	changed real constants to use dot syntax

*)
          
END_FUNCTION_BLOCK

FUNCTION_BLOCK CYCLE_TIME
  VAR_INPUT
    RST : BOOL;
  END_VAR
  VAR_OUTPUT
    ct_min : TIME;
    ct_max : TIME;
    ct_last : TIME;
    systime : TIME;
    sysdays : INT;
    cycles : DWORD;
  END_VAR
  VAR
    last_cycle : TIME;
    tx : TIME;
    init : BOOL;
  END_VAR

            tx := DWORD_TO_TIME(T_PLC_MS()) - last_cycle;
IF rst THEN
	ct_min := t#10h;
	ct_max := t#0ms;
	cycles := 0;
ELSIF last_cycle > t#0s THEN
	IF tx < ct_min THEN ct_min := tx;
	ELSIF tx > ct_max THEN ct_max := tx;
	END_IF;
	ct_last := tx;
ELSIF ct_min = t#0s THEN
	ct_min := t#0s - t#1ms;
END_IF;
IF init THEN
	systime := systime + tx;
		IF systime >= t#1d THEN
			systime := systime - t#1d;
			sysdays := sysdays + 1;
		END_IF;
END_IF;
init := TRUE;
last_cycle := last_cycle + tx;
cycles := cycles + 1;

(*	revision history
hm 12.12.2006		rev 1.1
	added cycles output, a dword cycle counter.
hm 10.3.2007			rev 1.2
	changed initialization of ct_min to t#10h for compatibility with siemens s7

hm	16.9.2007		rev 1.2
	changed Time() in T_PLC_MS() for compatibility resons

*)
          
END_FUNCTION_BLOCK

FUNCTION_BLOCK DT_SIMU
  VAR_INPUT
    START : DT;
    SPEED : REAL := 1;
  END_VAR
  VAR_OUTPUT
    DTS : DT;
  END_VAR
  VAR
    tc : DWORD;
    init : BOOL;
    last : DWORD;
    tx : DWORD;
    td : DWORD;
  END_VAR

            (* read system timer *)
tx := T_PLC_MS();
tc := REAL_TO_DWORD(DWORD_TO_REAL(tx - last) * speed);

IF NOT init THEN
	init := TRUE;
	DTS := Start;
	tc := 0;
	last := tx;
ELSIF SPEED = 0.0 THEN
	DTS := DWORD_TO_DT(DT_TO_DWORD(DTS) + 1);
ELSIF tc >= 1000 THEN
	td := (tc / 1000) * 1000;
	DTS := DTS + DWORD_TO_TIME(td);
	last := last + REAL_TO_DWORD(DWORD_TO_REAL(td) / speed);
END_IF;

(* revision history
hm	11. sep. 2008	rev 1.0
	original version

hm	16. nov	2008	rev 1.1
	added type conversions for compatibility reasons

hm	8.	mar. 2009	rev 1.2
	added increment by cycle mode

*)

          
END_FUNCTION_BLOCK

FUNCTION_BLOCK FLOW_METER
  VAR_INPUT
    VX : REAL;
    E : BOOL;
    RST : BOOL;
    {attribute 'input_constant'}
    PULSE_MODE : BOOL;
    {attribute 'input_constant'}
    UPDATE_TIME : TIME := TIME#1s0ms;
  END_VAR
  VAR_OUTPUT
    F : REAL;
  END_VAR
  VAR_IN_OUT
    X : REAL;
    Y : UDINT;
  END_VAR
  VAR
    tx : TIME;
    tl : TIME;
    int1 : INTEGRATE;
    init : BOOL;
    e_last : BOOL;
    tmp : INT;
    x_last : REAL;
    y_last : UDINT;
  END_VAR

            IF NOT init THEN	(* init on power up *)
	init := TRUE;
	tl := tx;
	x_last := X;
	y_last := Y;
	int1.K := 2.7777777777777777E-4;
END_IF;

(* run integrator *)
int1(E := NOT (RST OR PULSE_MODE) AND E, X := VX, Y := X);	(* gated operation *)

IF RST THEN		(* reset *)
	X := 0.0;
	Y := 0;
	tl := tx;
	x_last := 0.0;
	y_last := 0;
ELSIF E AND PULSE_MODE THEN	(* check for pulse mode *)
	IF NOT e_last THEN X := X + VX; END_IF;
END_IF;
e_last := E;

(* reduce X to be less than 1 and increase Y respectively *)
IF X > 1.0 THEN
	tmp := FLOOR(X);
	Y := Y + INT_TO_UDINT(tmp);
	X := X - INT_TO_REAL(tmp);
END_IF;

(* calculate the current flow *)
tx := DWORD_TO_TIME(T_PLC_MS());
IF tx - tl >= UPDATE_TIME AND UPDATE_TIME > t#0s THEN
	F := (UDINT_TO_REAL(Y - y_last) + X - x_last) / TIME_TO_REAL(tx - tl) * 3.6E6;
	y_last := Y;
	x_last := X;
	tl := tx;
END_IF;



(* revision history
hm	23. jan. 2011	rev 1.0
	original version

*)

          
END_FUNCTION_BLOCK

FUNCTION_BLOCK M_D
  VAR_INPUT
    start : BOOL;
    stop : BOOL;
    tmax : TIME := TIME#14400m0s0ms;
    rst : BOOL;
  END_VAR
  VAR_OUTPUT
    PT : TIME;
    ET : TIME;
    run : BOOL;
  END_VAR
  VAR
    edge : BOOL;
    T0 : TIME;
    tx : TIME;
    startup : BOOL;
  END_VAR

            (* check for rst input *)
IF rst OR et >= tmax THEN
	pt := t#0ms;
	et := t#0ms;
	startup := FALSE;
	run := FALSE;
END_IF;

(* avoid timers to start when input is true at startup *)
IF NOT startup THEN
	edge := start;
	startup := TRUE;
END_IF;

(* read system timer *)
tx := DWORD_TO_TIME(T_PLC_MS());

(* detect rising edge on start *)
IF start AND NOT edge AND NOT stop THEN
	t0 := tx;
	run := TRUE;
	pt := t#0s;
ELSIF stop AND run THEN
	pt := et;
	run := FALSE;
END_IF;
edge := start;
IF run THEN et := tx - t0; END_IF;

(* revision history
hm		2.5.2007	rev 1.0
	original version

hm		16.9.2007	rev 1.1
	changes time() to T_plc_ms() for compatibility reasons

hm	27. feb 2009	rev 1.2
	deleted unnecessary init with 0
*)

          
END_FUNCTION_BLOCK

FUNCTION_BLOCK M_T
  VAR_INPUT
    IN : BOOL;
    TMAX : TIME := TIME#14400m0s0ms;
    RST : BOOL;
  END_VAR
  VAR_OUTPUT
    PT : TIME;
    ET : TIME;
  END_VAR
  VAR
    edge : BOOL;
    start : TIME;
    tx : TIME;
  END_VAR

            (* read system time *)
tx := DWORD_TO_TIME(T_PLC_MS());

IF RST OR ET >= TMAX THEN
	PT :=  t#0s;
	ET := t#0s;
ELSIF IN THEN
	IF NOT edge THEN start := tx; END_IF;
	ET := tx - start;
ELSE
	PT := ET;
END_IF;
edge := IN;



(* revision history
hm	4. aug. 2006	rev 1.0
	original version

hm	2. may. 2007	rev 1.1
	added init variable to avoid unreasonable measurement if falling edge occurs first.
	added et (elapsed time) output to count from 0 at rising edge until a falling edge resets et to 0.
	added reset input.

hm	16. sep. 2007	rev 1.2
	changes time() to T_plc_ms() for compatibility reasons

hm	17. dec. 2008	rev 1.3
	code optimized

hm	10. mar. 2009	rev 1.4
	removed nested comments
	removed double assignments

*)
          
END_FUNCTION_BLOCK

FUNCTION_BLOCK M_TX
  VAR_INPUT
    in : BOOL;
    tmax : TIME := TIME#14400m0s0ms;
    rst : BOOL;
  END_VAR
  VAR_OUTPUT
    TH : TIME;
    TL : TIME;
    DC : REAL;
    F : REAL;
    ET : TIME;
  END_VAR
  VAR
    edge : BOOL;
    start : TIME;
    stop : TIME;
    tx : TIME;
    rise : BOOL;
    fall : BOOL;
    startup : BOOL;
  END_VAR

            (* check FOR rst input *)
IF rst OR (et >= tmax) THEN
	rise := FALSE;
	fall := FALSE;
	startup := FALSE;
	th := t#0ms;
	tl := t#0ms;
	DC := 0.0;
	F := 0.0;
	ET := t#0s;
END_IF;

(* avoid timers to start when input is true at startup *)
IF NOT startup THEN
	edge := in;
	startup := TRUE;
END_IF;

(* read system timer *)
tx := DWORD_TO_TIME(T_PLC_MS());

(* edge trigger rising and falling edge *)
IF in XOR edge THEN
	edge := in;
	(* rising edge starts measurement *)
	IF in THEN
		start := Tx;
		rise := TRUE;
		IF fall THEN tl := start - stop; END_IF;
		IF th > t#0ms AND tl > t#0ms THEN
			dc := TIME_TO_REAL(th) / TIME_TO_REAL(th+tl);
			f := 1000.0 / TIME_TO_REAL(th + tl);
		END_IF;
	(* falling edge starts second cycle measurement *)
	ELSE
		stop := Tx;
		fall := TRUE;
		IF rise THEN th := stop - start; END_IF;
		IF th > t#0ms AND tl > t#0ms THEN
			dc := TIME_TO_REAL(th) /  TIME_TO_REAL(th+tl);
			f := 1000.0 / TIME_TO_REAL(th + tl);
		END_IF;
	END_IF;
END_IF;
IF rise THEN et := tx - start; END_IF;

(* revision history
hm	4. aug. 2006	rev 1.0
	original version

hm	2. mai. 2007	rev 1.1
	made sure that no undefined values would be measured at startup conditions
	added output et
	added rst input
	added tmax input

hm	16. sep. 2007	rev 1.2
	changes time() to T_plc_ms() for compatibility reasons

hm	27. feb. 2009	rev 1.3
	deleted unnecessary init with 0

hm	11. mar. 2009	rev 1.4
	changed real constants to use dot syntax

*)
          
END_FUNCTION_BLOCK

FUNCTION_BLOCK METER
  VAR_INPUT
    M1 : REAL;
    M2 : REAL;
    I1 : BOOL;
    I2 : BOOL;
    D : REAL := 1;
    RST : BOOL;
  END_VAR
  VAR_IN_OUT
    MX : REAL;
  END_VAR
  VAR
    MR : REAL2;
    MX1 : REAL;  (* current consumption value on M1 and M2 *)
    MX2 : REAL;  (* current consumption value on M1 and M2 *)
    tx : DWORD;
    last : DWORD;
    tc : REAL;
    init : BOOL;
  END_VAR

            (* measure the last cycle time and make sure we onle execute once every millisecond *)
tx := T_PLC_MS();
IF NOT init THEN
	init := TRUE;
	last := tx;
	mr.RX := mx;
	mr.R1 := 0.0;
ELSIF tx = last THEN
	RETURN;
ELSE
	tc := DWORD_TO_REAL(tx - last) * 0.001;
END_IF;
last := tx;

(* reset *)
IF rst THEN
	mr.R1 := 0.0;
	mr.RX := 0.0;
ELSE
	(* current consumption measurement *)
	IF I1 THEN MX1 := M1; ELSE MX1 := 0.0; END_IF;
	IF I2 THEN MX2 := M2; ELSE MX2 := 0.0; END_IF;
	(* add up the current values in a double real *)
	MR := R2_ADD(MR,(SEL(I1,0.0,mx1) + SEL(I2, 0.0, mx2)) / D * TC);
	(* set the current output value *)
	MX := mr.RX;
END_IF;




(* revision history

hm	16. sep.2007		rev 1.0
	original version

hm	7. feb 2008		rev 1.1
	use new version of ft_int to avoid a counting stop at high values
	deleted unnecessary limits

hm	24. mar. 2008	rev 1.2
	use data_type real2 to extend accuracy to 15 digits total
	do not use ft_int which adds unnecessary overhead

hm	8. feb. 2009	rev 1.3
	changed mx to be I/O
	make sure calculation works for cycle times < 1 ms

hm	8. mar. 2009	rev 1.4
	last was not updated
	code improvements

*)

          
END_FUNCTION_BLOCK

FUNCTION_BLOCK METER_STAT
  VAR_INPUT
    IN : REAL;
    DI : DATE;
    RST : BOOL;
  END_VAR
  VAR_IN_OUT
    Last_Day : REAL;
    Current_Day : REAL;
    Last_Week : REAL;
    Current_Week : REAL;
    Last_Month : REAL;
    Current_Month : REAL;
    Last_Year : REAL;
    Current_Year : REAL;
  END_VAR
  VAR RETAIN
    Year_Start : REAL;
    Month_Start : REAL;
    Week_Start : REAL;
    Day_Start : REAL;
    last_run : DATE;
  END_VAR

            IF rst THEN
	Last_Day := 0.0;
	Current_Day := 0.0;
	Day_start := IN;
	Last_week := 0.0;
	Current_week := 0.0;
	Week_start := in;
	Last_month := 0.0;
	Current_month := 0.0;
	month_start := in;
	last_year := 0.0;
	current_year := 0.0;
	year_start := in;
ELSE
	Current_Day := IN - Day_Start;
	Current_Week := In - Week_Start;
	Current_Month := IN - Month_Start;
	Current_Year := IN - Year_Start;
END_IF;

IF YEAR_OF_DATE(DI) > YEAR_OF_DATE(last_run) THEN
	(* a new year has started *)
	last_year := current_year;
	current_year := 0.0;
	year_start := in;
	last_month := current_month;
	current_month := 0.0;
	month_start := in;
	last_day := current_day;
	current_day := 0.0;
	day_start := in;
ELSIF MONTH_OF_DATE(DI) > MONTH_OF_DATE(last_run) THEN
	(* a new month has started, january is alrerady done by year change *)
	last_month := current_month;
	current_month := 0.0;
	month_start := in;
	last_day := current_day;
	current_day := 0.0;
	day_start := in;
ELSIF DAY_OF_YEAR(di) > DAY_OF_YEAR(last_run) THEN
	(* day has chaged, first day of year and first day of month has already been taken care of *)
	last_day := current_day;
	current_day := 0.0;
	day_start := in;
END_IF;
IF DAY_OF_WEEK(DI) < DAY_OF_WEEK(last_run) THEN
	(* a new week has started *)
	last_week := current_week;
	current_week := 0.0;
	week_start := in;
END_IF;
last_run := di;

(* revision history
hm	16. sep. 2007	rev 1.0
	original version

hm	7. oct. 2008	rev 1.1
	changed function year_to_year_of_date
	changed function month to month_of_date
	changed function weekday to day_of_week

hm	11. mar. 2009	rev 1.2
	changed real constants to use dot syntax

hm	18. jul. 2009	rev 1.3
	changes all outputs to be I/O
*)

          
END_FUNCTION_BLOCK

FUNCTION_BLOCK ONTIME
  VAR_INPUT
    IN : BOOL;
    RST : BOOL;
  END_VAR
  VAR_IN_OUT
    SECONDS : UDINT;
    CYCLES : UDINT;
  END_VAR
  VAR
    tx : DWORD;
    last : DWORD;
    edge : BOOL;
    init : BOOL;
    ms : DWORD;
  END_VAR

            (* read system time *)
tx := T_PLC_MS();

(* make sure the first cycle works correctly *)
IF NOT init OR rst THEN
	init := TRUE;
	last := tx;
	ms := 0;
ELSIF RST THEN
	SECONDS := 0;
	CYCLES := 0;
ELSIF IN THEN
	(* add the current milliseconds *)
	ms := (tx - last) + ms;
	IF ms >= 1000 THEN
		seconds := seconds + 1;
		ms := ms - 1000;
	END_IF;
	cycles := cycles + BOOL_TO_UINT(NOT edge);
END_IF;
last := tx;
edge := in;


(* revision history
hm 22.2.2007		rev 1.1
	changed VAR RETAIN PERSISTENT to VAR RETAIN for better compatibility
	wago lon contollers do not support persisitent

hm 2.8.2007		rev 1.2
	adding time up in a real number will automatically lead to the point where 
	small time scales like the cycle time will be below the resolution of real and therefore
	ontime would not increase in small steps as necessary
	the time is now measured internally in two  dwords and be converted to real only for
	output purposes.
	deleted the variable power because it was unnecessary

hm	16.9.2007		rev 1.3
	changes time() to T_plc_ms() for compatibility reasons

hm	2. dec. 2007	rev 1.4
	chaged code for better performance

hm	16. mar. 2008	rev 1.5
	added type conversions to avoid warnings under codesys 3.0

hm	21. oct. 2008	rev 2.0
	changed module for much better performance and allow for external result storage

hm	10. nov. 2008	rev 2.1
	increased internal resolution to milliseconds

hm	16. nov. 2008	rev 2.2
	changed typecast to avoid warnings

hm	17. dec. 2008	rev 2.3
	fixed an error when in would be true for more then 49 days

hm	17. jan 2011	rev 2.4
	init will not clear seconds and cycles, only rst clears these values	

*)
          
END_FUNCTION_BLOCK

FUNCTION T_PLC_MS : DWORD
  VAR CONSTANT
    debug : BOOL := 0;
    N : INT := 0;
    offset : DWORD := 0;
  END_VAR
  VAR
    tx : TIME;
  END_VAR

            tx := TIME();
T_PLC_MS := TIME_TO_DWORD(Tx);
(* hier muss die korrektur für step7 stattfinden
plctime muss den vollen wertebereich von time ausnutzen:
wenn bei step7 time -24tage bis plus 24 tage ist dann muss der timer auch beim überlauf auf -24tage springen 
und auf keinen fall auf 0 !!!!
für siemens muss ein weiterer fb im main eingebunden werden der sicherstellt das alle 32 bits durchgezählt werden.
es kann nur ein fb sein den er muss sich das oberste (32te) bit merken.
oder etwa spring s7 bei überlauf auf -24 tage????? dann wäre keine korrektur nötig.
*)
IF debug THEN
	T_PLC_MS := (SHL(T_PLC_MS,N) OR SHL(DWORD#1,N)-1) + OFFSET;
END_IF;

(* revision history
hm	14.9.2007	rev 1.0
	original version

hm	12. nov 2007	rev 1.1
	added temporaray variable tx because some compilers could not handle time() as an argument

hm	16. nov. 2008	rev 1.2
	initialized constants with 0 for compatibility reasons
*)
          
END_FUNCTION

FUNCTION T_PLC_US : DWORD
  VAR CONSTANT
    debug : BOOL := 0;
    N : INT := 0;
    offset : DWORD := 0;
  END_VAR
  VAR
    tx : TIME;
  END_VAR

            tx := TIME();
T_PLC_US := TIME_TO_DWORD(Tx)*1000;
(* hier muss die korrektur für step7 stattfinden
plctime muss den vollen wertebereich von time ausnutzen:
wenn bei step7 time -24tage bis plus 24 tage ist dann muss der timer auch beim überlauf auf -24tage springen 
und auf keinen fall auf 0 !!!!
für siemens muss ein weiterer fb im main eingebunden werden der sicherstellt das alle 32 bits durchgezählt werden.
es kann nur ein fb sein den er muss sich das oberste (32te) bit merken.
oder etwa spring s7 bei überlauf auf -24 tage????? dann wäre keine korrektur nötig.
*)
IF debug THEN
	T_PLC_US := (SHL(T_PLC_US,N) OR SHL(DWORD#1,N)-1) + OFFSET;
END_IF;

(* revision history
hm	14.9.2007	rev 1.0
	original version

hm	12. nov 2007	rev 1.1
	added temporaray variable tx because some compilers could not handle time() as an argument

hm	16. nov. 2008	rev 1.2
	initialized constants with 0 for compatibility reasons

*)
          
END_FUNCTION

FUNCTION_BLOCK TC_MS
  VAR_OUTPUT
    TC : DWORD;
  END_VAR
  VAR
    init : BOOL;
    tx : DWORD;
    last : DWORD;
  END_VAR

            (* read system timer *)
tx := T_PLC_MS();

IF NOT init THEN
	init := TRUE;
	TC := 0;
ELSE
	tc := tx - last;
END_IF;
last := tx;

(* revision history
hm		13. mar. 2008	rev 1.0
	original version

*)

          
END_FUNCTION_BLOCK

FUNCTION_BLOCK TC_S
  VAR_OUTPUT
    TC : REAL;
  END_VAR
  VAR
    init : BOOL;
    tx : DWORD;
    last : DWORD;
  END_VAR

            (* read system timer *)
tx := T_PLC_US();

IF NOT init THEN
	init := TRUE;
	TC := 0.0;
ELSE
	tc := DWORD_TO_REAL(tx - last)*1.0E-6;
END_IF;
last := tx;

(* revision history
hm	13. mar. 2008	rev 1.0
	original version

hm	16. mar 2008	rev 1.1
	added type conversion to avoid warnings under codesys 3.0

hm	11. mar. 2009	rev 1.2
	changed real constants to use dot syntax

*)

          
END_FUNCTION_BLOCK

FUNCTION_BLOCK TC_US
  VAR_OUTPUT
    TC : DWORD;
  END_VAR
  VAR
    init : BOOL;
    tx : DWORD;
    last : DWORD;
  END_VAR

            (* read system timer *)
tx := T_PLC_US();

IF NOT init THEN
	init := TRUE;
	TC := 0;
ELSE
	tc := tx - last;
END_IF;
last := tx;

(* revision history
hm		13. mar. 2008	rev 1.0
	original version

*)

          
END_FUNCTION_BLOCK

FUNCTION MULTI_IN : REAL
  VAR_INPUT
    in_1 : REAL;
    in_2 : REAL;
    in_3 : REAL;
    default : REAL;
    in_min : REAL;
    in_max : REAL;
    mode : BYTE;
  END_VAR
  VAR
    count : INT;
    F1 : BOOL;
    F2 : BOOL;
    F3 : BOOL;
  END_VAR

            F1 :=  in_1 > in_min AND in_1 < in_max;
F2 :=  in_2 > in_min AND in_2 < in_max;
F3 :=  in_3 > in_min AND in_3 < in_max;

CASE mode OF
0:	count := 0;
	IF F1 THEN
		count := count + 1;
		MULTI_IN := in_1;
	ELSE
		MULTI_IN := 0.0;
	END_IF;
	IF F2 THEN
		count := count + 1;
		MULTI_IN := MULTI_IN + in_2;
	END_IF;
	IF F3 THEN
		count := count + 1;
		MULTI_IN := MULTI_IN + in_3;
	END_IF;
	MULTI_IN := SEL(count = 0, MULTI_IN / INT_TO_REAL(count), default);

1:	MULTI_IN := SEL(F1, default, IN_1);

2:	MULTI_IN := SEL(F2, default, IN_2);

3:	MULTI_IN := SEL(F3, default, IN_3);

4:	MULTI_IN := default;

5:	MULTI_IN := SEL(F1, in_max, IN_1);
	IF F2 AND in_2 < MULTI_IN THEN MULTI_IN := in_2; END_IF;
	IF F3 AND in_3 < MULTI_IN THEN MULTI_IN := in_3; END_IF;
	IF MULTI_IN = in_max THEN MULTI_IN := default; END_IF;

6:	MULTI_IN := SEL(F1, in_min, IN_1);
	IF F2 AND in_2 > MULTI_IN THEN MULTI_IN := in_2; END_IF;
	IF F3 AND in_3 > MULTI_IN THEN MULTI_IN := in_3; END_IF;
	IF MULTI_IN = in_min THEN MULTI_IN := default; END_IF;

7:	IF F1 AND F2 AND F3 THEN MULTI_IN := MID3(in_1, in_2, in_3);
	ELSIF F1 AND F2 THEN MULTI_IN := MIN(in_1, in_2);
	ELSIF F1 AND F3 THEN MULTI_IN := MIN(in_1, in_3);
	ELSIF F2 AND F3 THEN MULTI_IN := MIN(in_2, in_3);
	ELSIF F1 THEN MULTI_IN := in_1;
	ELSIF F2 THEN MULTI_IN := in_2;
	ELSIF F3 THEN MULTI_IN := in_3;
	ELSE MULTI_IN := default;
	END_IF;

END_CASE;

(*
hm 1.1.2007		rev 1.1
	changed midr to mid3 function

hm	14. 10. 2008	rev 1.2
	corrected an error for in_3 overrange detection
	improved performance

hm	11. mar. 2009	rev 1.3
	changed real constants to use dot syntax

hm	18. jul. 2009	rev 1.4
	improved performance
*)
          
END_FUNCTION

FUNCTION RES_NI : REAL
  VAR_INPUT
    T : REAL;
    R0 : REAL;
  END_VAR
  VAR CONSTANT
    A : REAL := 0.5485;
    B : REAL := 0.000665;
    C : REAL := 2.805E-09;
  END_VAR
  VAR
    T2 : REAL;
  END_VAR

            T2 := T * T;
RES_NI := R0 + A * T + B * T2 + C * T2 * T2;

(* revision history

hm	4.8.2006		rev 1.0
	original version

hm	13.9.2007		rev 1.1
	changed coding for better performance

hm	2. dec. 2007	rev 1.2
	changed code for better performance
*)

(*

 Auszug aus DIN 43760 für Ni100

°C		R		°C		R		°C	R		°C		R		°C		R

-60 	69,5 	-10 	94,6 	40 	123,0 	90 		154,9 	140 	190,9
-55 	71,9 	-5 		97,3 	45 	126,0 	95 		158,3 	145 	194,8
-50 	74,3 	0 		100,0 	50 	129,1 	100 	161,8 	150 	198,7
-45 	76,7 	5 		102,8 	55 	132,2 	105 	165,3 	155 	202,6
-40 	79,1 	10 		105,6 	60 	135,3 	110 	168,8 	160 	206,6
-35 	81,6 	15 		108,4 	65 	138,5 	115 	172,4 	165 	210,7
-30 	84,2 	20 		111,2 	70 	141,7 	120 	176,0 	170 	214,8
-25 	86,7 	25 		114,1 	75 	145,0 	125 	179,6 	175 	219,0
-20 	89,3 	30 		117,1 	80 	148,3 	130 	183,3 	180 	223,2
-15 	91,9 	35 		120,0 	85 	151,6 	135 	187,1 	  	 

